// SIMATIC STEP 7 (V5.x) project BIW01_2012
// CPU: CPU 416-2 DP
// station: Hardware
// station: PLC1
// station: P_ADR_BUS
// program: GCPRO_Import
// program: Current400
// program: tmpGP-BIB
// program: tmpMH-BIB
// program: Current
// program: S7-Programm
// program: Baustein Kopie
// program: AG_Abzug
// program: temp
// program: temp2

SYMBOL_TABLE
"SYS_CBitDB"	DB 2	DB 2	// SYS: Changebit interface
"SYS_DirectCtrlDB"	DB 3	DB 3	// GCS7: PC direct control interface default DB
"SYS_HornDB"	DB 4	DB 4	// GCS7: Data Horn Modul
"SYS_LOG_Queue"	DB 5	DB 5	// PC Interface to log
"GCS7_GrCtrlDBTmp"	DB 6	FB 9	// Class date of FB9
"GCS7_RS485CtrlDB"	DB 7	FB 7	// GCS7: Communication controller opto22
"GCS7_ScaleControlDB"	DB 8	DB 8	// GCS7: Scale control buffer
"GCS7_GrCtrlDB"	DB 9	DB 9	// GCS7: Group control buffer
"SYS_DirectCtrlLCDB"	DB 10	DB 10	// GCS7: PC Direct Control Interface Remote Parameter
"TEST_IOSimuliInput"	DB 16	DB 16	// TEST: Only for serial (MPI) simulation
"TEST_IOSimuliOutput"	DB 17	DB 17	// TEST: Only for serial (MPI) simulation
"KebaHT4Data"	DB 20	FB 80	// Data KebaHT4Data
"SYS_PCCDirectCtrlDB"	DB 40	DB 40	// SYS: PC direct control interface PIC / WinCos /MELE
"SYS_PC1DirectCtrlDB"	DB 41	DB 41	// SYS: PC direct control interface pcc 1 (WinCC)
"SYS_PC2DirectCtrlDB"	DB 42	DB 42	// SYS: PC direct control interface pcc 2 (WinCC)
"SYS_PC3DirectCtrlDB"	DB 43	DB 43	// SYS: PC direct control interface pcc 1 (WinCC)
"SYS_PC4DirectCtrlDB"	DB 44	DB 44	// SYS: PC direct control interface pcc 4 (WinCC)
"SYS_PC5DirectCtrlDB"	DB 45	DB 45	// SYS: PC direct control interface pcc 5 (WinCC)
"SYS_PC6DirectCtrlDB"	DB 46	DB 46	// SYS: PC direct control interface pcc 6 (WinCC)
"SYS_PC7DirectCtrlDB"	DB 47	DB 47	// SYS: PC direct control interface pcc 7 (WinCC)
"SYS_ObjViewDirectCtrlDB"	DB 48	DB 48	// SYS: PC direct control interface for ObjView
"SYS_IHTestDirectCtrlDB"	DB 49	DB 49	// SYS: PC direct control interface for inhouse test
"PLC_SystemDB"	DB 50	DB 50	// PLC: System informations
"PLC_DPInfo"	DB 51	DB 51	// Summary Slave errors
"SSA_SYS_ASI_Info"	DB 52	DB 52	// Summary Slave errors
"PC_StorageDB"	DB 53	DB 53	// PC: Storage with free assignment
"ASW_TimerSettings"	DB 56	DB 56	// ASW: Timer settings
"ASW_Counter"	DB 57	DB 57	// ASW: Counter presettings
"SYS_PC1CBitDB"	DB 61	UDT 10020	// SYS: Changebit interface pcc 1 | PIC.LCT | MELE
"SYS_PC2CBitDB"	DB 62	UDT 10020	// SYS: Changebit interface pcc 2 | PIC.LMX
"SYS_PC3CBitDB"	DB 63	UDT 10020	// SYS: Changebit interface pcc 3
"SYS_PC4CBitDB"	DB 64	UDT 10020	// SYS: Changebit interface pcc 4
"GCS7_EREDB"	DB 71	FB 71	// GCS7: ERE
"SYS_DPInfoM1"	DB 75	FB 76	// SYS: PROFIBUS-DP diagnostic master 1
"SYS_DPInfoM2"	DB 76	FB 76	// SYS: PROFIBUS-DP diagnostic master 2
"SYS_DPInfoM3"	DB 77	FB 76	// SYS: PROFIBUS-DP diagnostic master 3
"SYS_DPInfoM4"	DB 78	FB 76	// SYS: PROFIBUS-DP diagnostic master 4
"PLC_BinListDB"	DB 79	FB 79	// Central bin list DB
"ASW_GraphicData"	DB 80	DB 80	// Win CC animation: Ways, function key, plant parameter
"ASW_PlantParData"	DB 81	DB 81	// Plant parameters and data time
"PCC_Data4"	DB 84	DB 84	// WinCC/PIC
"PCC_Data5"	DB 85	DB 85	// WinCC/PIC
"PCC_Data6"	DB 86	DB 86	// WinCC/PIC
"PCC_Data7"	DB 87	DB 87	// WinCC/PIC
"PCC_Data8"	DB 88	DB 88	// WinCC/PIC
"PCC_Data9"	DB 89	DB 89	// WinCC/PIC
"PCC_YieldScaleDB"	DB 90	DB 90	// PCC: Databuffer for PCC yield calculation
"COM_RS485Loop1DB"	DB 91	FB 7	// COM: RS485 loop1 scales and MYEB
"COM_RS485Loop2DB"	DB 92	FB 7	// COM: RS485 loop2 roolers
"COM_RS485Loop3DB"	DB 93	FB 7	// COM: RS485 loop3
"COM_RS485Loop4DB"	DB 94	FB 7	// COM: RS485 loop4
"SYS_SimpleDPInfo4DB"	DB 98	DB 98	// Data DP Diagnose
"SYS_StartWarningDB"	DB 100	FB 100	// SYS:  Startwarning modul
"ASW_DFCATargData"	DB 480	DB 480	// ASW_DFCATargData
"PLC1Snd"	DB 1711	DB 1711	// COM: Send data to PLC 1
"PLC2Snd"	DB 1712	DB 1712	// COM: Send data to PLC 2
"PLC3Snd"	DB 1713	DB 1713	// COM: Send data to PLC 3
"PLC4Snd"	DB 1714	DB 1714	// COM: Send data to PLC 4
"PLC5Snd"	DB 1715	DB 1715	// COM: Send data to PLC 5
"PLC6Snd"	DB 1716	DB 1716	// COM: Send data to PLC 6
"PLC7Snd"	DB 1717	DB 1717	// COM: Send data to PLC 7
"PLC8Snd"	DB 1718	DB 1718	// COM: Send data to PLC 8
"PLC9Snd"	DB 1719	DB 1719	// COM: Send data to PLC 9
"PLC1Rcv"	DB 1721	DB 1721	// COM: Receive data from PLC 1
"PLC2Rcv"	DB 1722	DB 1722	// COM: Receive data from PLC 2
"PLC3Rcv"	DB 1723	DB 1723	// COM: Receive data from PLC 3
"PLC4Rcv"	DB 1724	DB 1724	// COM: Receive data from PLC 4
"PLC5Rcv"	DB 1725	DB 1725	// COM: Receive data from PLC 5
"PLC6Rcv"	DB 1726	DB 1726	// COM: Receive data from PLC 6
"PLC7Rcv"	DB 1727	DB 1727	// COM: Receive data from PLC 7
"PLC8Rcv"	DB 1728	DB 1728	// COM: Receive data from PLC 8
"PLC9Rcv"	DB 1729	DB 1729	// COM: Receive data from PLC 9
"PLC10Snd"	DB 1730	DB 1730	// COM: Send data to PLC 10
"PLC11Snd"	DB 1731	DB 1731	// COM: Send data to PLC 11
"PLC12Snd"	DB 1732	DB 1732	// COM: Send data to PLC 12
"PLC13Snd"	DB 1733	DB 1733	// COM: Send data to PLC 13
"PLC14Snd"	DB 1734	DB 1734	// COM: Send data to PLC 14
"PLC15Snd"	DB 1735	DB 1735	// COM: Send data to PLC 15
"PLC16Snd"	DB 1736	DB 1736	// COM: Send data to PLC 16
"PLC10Rcv"	DB 1740	DB 1740	// COM: Receive data from PLC 10
"PLC11Rcv"	DB 1741	DB 1741	// COM: Receive data from PLC 11
"PLC12Rcv"	DB 1742	DB 1742	// COM: Receive data from PLC 12
"PLC13Rcv"	DB 1743	DB 1743	// COM: Receive data from PLC 13
"PLC14Rcv"	DB 1744	DB 1744	// COM: Receive data from PLC 14
"PLC15Rcv"	DB 1745	DB 1745	// COM: Receive data from PLC 15
"PLC16Rcv"	DB 1746	DB 1746	// COM: Receive data from PLC 16
"ComPLC1Snd"	DB 1761	FB 1701	// COM: Send buffer PLC 1
"ComPLC2Snd"	DB 1762	FB 1701	// COM: Send buffer PLC 2
"ComPLC3Snd"	DB 1763	FB 1701	// COM: Send buffer PLC 3
"ComPLC4Snd"	DB 1764	FB 1701	// COM: Send buffer PLC 4
"ComPLC5Snd"	DB 1765	FB 1701	// COM: Send buffer PLC 5
"ComPLC6Snd"	DB 1766	FB 1701	// COM: Send buffer PLC 6
"ComPLC7Snd"	DB 1767	FB 1701	// COM: Send buffer PLC 7
"ComPLC8Snd"	DB 1768	FB 1701	// COM: Send buffer PLC 8
"ComPLC9Snd"	DB 1769	FB 1701	// COM: Send buffer PLC 9
"ComPLC1Rcv"	DB 1771	FB 1702	// COM: Receive buffer PLC 1
"ComPLC2Rcv"	DB 1772	FB 1702	// COM: Receive buffer PLC 2
"ComPLC3Rcv"	DB 1773	FB 1702	// COM: Receive buffer PLC 3
"ComPLC4Rcv"	DB 1774	FB 1702	// COM: Receive buffer PLC 4
"ComPLC5Rcv"	DB 1775	FB 1702	// COM: Receive buffer PLC 5
"ComPLC6Rcv"	DB 1776	FB 1702	// COM: Receive buffer PLC 6
"ComPLC7Rcv"	DB 1777	FB 1702	// COM: Receive buffer PLC 7
"ComPLC8Rcv"	DB 1778	FB 1702	// COM: Receive buffer PLC 8
"ComPLC9Rcv"	DB 1779	FB 1702	// COM: Receive buffer PLC 9
"ComPLC10Snd"	DB 1780	FB 1701	// COM: Send buffer PLC 10
"ComPLC11Snd"	DB 1781	FB 1701	// COM: Send buffer PLC 11
"ComPLC12Snd"	DB 1782	FB 1701	// COM: Send buffer PLC 12
"ComPLC13Snd"	DB 1783	FB 1701	// COM: Send buffer PLC 13
"ComPLC14Snd"	DB 1784	FB 1701	// COM: Send buffer PLC 14
"ComPLC15Snd"	DB 1785	FB 1701	// COM: Send buffer PLC 15
"ComPLC16Snd"	DB 1786	FB 1701	// COM: Send buffer PLC 16
"ComPLC10Rcv"	DB 1790	FB 1702	// COM: Receive buffer PLC 7
"ComPLC11Rcv"	DB 1791	FB 1702	// COM: Receive buffer PLC 1
"ComPLC12Rcv"	DB 1792	FB 1702	// COM: Receive buffer PLC 2
"ComPLC13Rcv"	DB 1793	FB 1702	// COM: Receive buffer PLC 3
"ComPLC14Rcv"	DB 1794	FB 1702	// COM: Receive buffer PLC 4
"ComPLC15Rcv"	DB 1795	FB 1702	// COM: Receive buffer PLC 5
"ComPLC16Rcv"	DB 1796	FB 1702	// COM: Receive buffer PLC 6
"SSA_VIS_Filter"	DB 2010	DB 2010	// Filter DB to convert Status for Viscontrol
"SIEMENS_READ"	FB 3	FB 3	// SIEMENS: FMS.read services with SIMATIC NET CPs
"SIEMENS_WRITE"	FB 6	FB 6	// SIEMENS: FMS.write services with SIMATIC NET CPs
"GCS7_RS485Ctrl"	FB 7	FB 7	// GCS7: Communication controller opto22
"GCS7_GrpCtrlMain"	FB 9	FB 9	// GCS7: Group control main program
"GCS7_GrpCtrlSub"	FB 10	FB 10	// GCS7: Group control subroutines
"GCS7_E_DigOutput"	FB 11	FB 11	// GCS7: Element digital output
"GCS7_E_Motor"	FB 12	FB 12	// GCS7: Element motor
"GCS7_E_ValveControl"	FB 13	FB 13	// GCS7: Element valve control
"GCS7_E_DigInput"	FB 14	FB 14	// GCS7: Element digital input continuous
"GCS7_E_PressureRange"	FB 16	FB 16	// GCS7: Element pressure range
"GCS7_E_AnalogOutput"	FB 17	FB 17	// GCS7: Element analog output
"GCS7_E_ATV"	FB 18	FB 18	// Element Control FU Altivar with Profibus
"GCS7_E_AnalogInput"	FB 19	FB 19	// GCS7: Element analog input
"GCS7_E_ValveControl4Pos"	FB 20	FB 20	// GCS7: Element valve control with 4 positions
"GCS7_E_DMDS"	FB 21	FB 21	// GCS7: Element DMDS
"GCS7_E_MZMN"	FB 22	FB 22	// GCS7: Element MZMN micro dosing
"GCS7_E_MYEB"	FB 23	FB 23	// GCS7: Element MYEB moisture control unit
"GCS7_E_MOZE"	FB 24	FB 24	// GCS7: Element MOZE water doser
"GCS7_E_MessageCtrl"	FB 25	FB 25	// GCS7: Element Control Message
"GCS7_E_DFCO"	FB 26	FB 26
"GCS7_E_MEAF_Bag"	FB 27	FB 27	// GCS7: Element Control MEAF-Bag with DP or OPTO22
"GCS7_E_FBAL"	FB 28	FB 28	// GCS7: Element Control Message
"GCS7_E_Sampler"	FB 29	FB 29	// GCS7: Element sampler MZER
"GCS7_E_Maintanance1"	FB 30	FB 30	// GCS7: Element Control Message
"GCS7_E_Maintanance2"	FB 31	FB 31	// GCS7: Element Control Message
"GCS7_E_MZAF"	FB 32	FB 32	// GCS7: Element MZAF flowbalancer
"GCS7_E_MYAH"	FB 33	FB 33	// GCS7: Element MYAH Yield PC
"GCS7_E_MYFC_MOZF"	FB 34	FB 34	// GCS7: Element MYFC/MOZF
"GCS7_E_MDDx"	FB 35	FB 35	// GCS7 Element MDDx Opto22 Communication
"GCS7_E_MYRA_MDEx"	FB 36	FB 36	// GCS7: Element MYRA/MDEF
"GCS7_E_MDDx_DP"	FB 37	FB 37	// SSW: Element MDDR/T Profibus Communication
"GCS7_E_DEVC"	FB 38	FB 38	// GCS7: Element MEAF Dev Control
"GCS7_E_MYFA_MOZD"	FB 39	FB 39	// GCS7: Element MYFA/MOZD automatic dampener
"GCS7_E_Scale"	FB 40	FB 40	// GCS7: Element scale control MWEE, MWEG,
"GCS7_M_MYFA"	FB 41	FB 41	// GCS7: Machine MYFA
"GCS7_E_BSPB"	FB 42	FB 42	// Vertikalschleifer
"GCS7_E_DCOS"	FB 43	FB 43	// GCS7: Element Control Dosing Control System
"GCS7_M_Scourer"	FB 44	FB 44	// GCS7: Machine scourer MHXF
"GCS7_M_Roll4Stand"	FB 45	FB 45	// GCS7: Machine 4 roll stand
"GCS7_M_Roll8Stand"	FB 46	FB 46	// GCS7: Machine 8 roll stand
"GCS7_M_PelletCooler"	FB 47	FB 47	// GCS7: Machine pellet cooler
"GCS7_M_Motors3W2HL"	FB 48	FB 48	// GCS7: Machine 3 Motors and 2 high levels
"GCS7_M_MDDX"	FB 49	FB 49	// GCS7: Machine Newtronic Roll Stand
"GCS7_M_Motor6Mon"	FB 50	FB 50	// GCS7: Machine motor with 6 monitoring elements
"GCS7_M_Motor2Mon"	FB 51	FB 51	// GCS7: Machine motor with 2 monitoring elements
"GCS7_M_MotorBypass"	FB 52	FB 52	// GCS7: Machine motor with bypass
"GCS7_M_Hopper"	FB 53	FB 53	// GCS7: Machine hopper
"GCS7_M_Mixer"	FB 54	FB 54	// GCS7: Machine mixer
"GCS7_M_DFZK"	FB 55	FB 55	// GCS7 Machine DFZK Vertical Rotor Mill
"GCS7_M_Discharger"	FB 56	FB 56	// GCS7: Machine discharger A
"GCS7_E_MTRI"	FB 57	FB 57	// GCS7: Element MTRI Remote Control
"GCS7_M_BCFA"	FB 58	FB 58	// GCS7: Machine Flaker Control System
"GCS7_M_DischargerMZAx"	FB 59	FB 59	// GCS7: Machine discharger with MZAF
"GCS7_M_Aspiration"	FB 60	FB 60	// GCS7: Machine aspiration
"GCS7_M_DPScaleMWBL_MWBS"	FB 61	FB 61	// GCS7: Machine MWBL/MWBS (Profibus+ Opto22)
"GCS7_M_DriveCurrent"	FB 62	FB 62	// GCS7: Machine DriveCurrent
"GCS7_M_DFCA"	FB 63	FB 63	// GCS7: Machine DFCA
"GCS7_M_MYFB"	FB 64	FB 64	// GCS7: Machine MYFB automatic dampener
"GCS7_M_PulsePhaseConv"	FB 65	FB 65	// GCS7: Machine pulse phase conveying system
"GCS7_M_Flift1Airlock"	FB 66	FB 66	// GCS7: Machine fluidlift with 1 airlock
"GCS7_M_Flift2Airlock"	FB 67	FB 67	// GCS7: Machine fluidlift with 2 airlocks
"GCS7_M_PressureVessel"	FB 68	FB 68	// GCS7 Machine Pressure Vessel Conveying
"GCS7_M_RotaryDis"	FB 69	FB 69	// GCS7: Machine rotary distributer
"GCS7_AddWayPattern"	FB 70	FB 70	// GCS7: Old and new waypattern are active
"GCS7_E_MaintananceCnt"	FB 71	FB 71	// GCS7: Maintanance Counter
"GCS7_E_DFCA_Com"	FB 73	FB 73	// GCS7: Communication DFCA pellet press
"GCS7_E_DFCA_Log"	FB 74	FB 74	// GCS7: Log when modify a parameter
"SYS_DP-Diagnosis"	FB 76	FB 76	// SIEMENS_DP-Diagnosis
"GCS7_ULQueue"	FB 77	FB 77
"GCS7_Bin"	FB 78	FB 78	// Functionality of a bin
"PLC_BinList"	FB 79	FB 79	// Central bin list
"KebaHT4"	FB 80	FB 80	// MAINTENANCE MOTOR CONTROL "HT4"
"GCS7_M_RGRP"	FB 81	FB 81	// GCS7: Machine RGRP
"GCS7_M_FluidlifVessel"	FB 82	FB 82	// GCS7 Machine Fluidlift with Pressure Vessel
"GCS7_E_Level"	FB 84	FB 84	// Level: Subtype of FB14
"GCS7_LiftingDevice"	FB 85	FB 85	// de: Hubzug
"GCS7_TractionDrive"	FB 86	FB 86	// Traction drive  de: Fahrantrieb
"GCS7_M_Roll8Stand_DP"	FB 87	FB 87	// SS: Machine 4/8 roll stand wit profibus
"GCS7_Ma_DischagerFlat"	FB 88	FB 88	// Machine Flat-bottom discharger
"STD_LineSecStdSub2"	FB 90	FB 90	// STD: Line and section control standard subroutines
"SYS_DPMultiDPInfo"	FB 98	FB 98	// SimpleMultiDPInfo
"SYS_DPDiagnostic"	FB 99	FB 99	// SYS: DP diagnostic and monitoring
"GCS7_StartWarning"	FB 100	FB 100	// GCS7 Start Warning Modul
"Gr050_Code"	FB 150	FB 150	// Group-FB  Machine FB44, FB47, FB50, FB51, FB52, FB56
"STD_StartupBinTime"	FB 801	FB 801	// STD: Startup bin filling procedure
"SSA_PneumaticControl_Fct"	FB 841	FB 841	// SSA: Pneumatic controller
"SSW_EL_ASI_Fct"	FB 899	FB 899	// Element Control ASI Master Wago/Profibus
"COM_PLCSend"	FB 1701	FB 1701	// COM: Send data to an other PLC
"COM_PLCReceive"	FB 1702	FB 1702	// COM: Receive data from an other PLC
"STD_PLCWatchdog"	FB 1703	FB 1703	// STD: PLC to PLC communication watchdog
"COM_Modbus_CMV96"	FB 1709	FB 1709	// Modbus interface to CMV96
"SSA_EL_Sampler_RFID"	FB 1714	FB 1714	// Baumer RFID
"SYS_CBitCtrl"	FC 2	FC 2	// SYS: Call change bit controller
"SYS_DirectCtrl"	FC 3	FC 3	// GCS7: PC direct control subroutines
"SYS_Horn_Code"	FC 4	FC 4	// GCS7: Code Horn Modul
"AG_SEND"	FC 5	FC 5	// Send Function for SEND-/RECEIVE-Services to SIMATIC NET CPs
"AG_RECEIVE"	FC 6	FC 6	// Receive Function for SEND-/RECEIVE-Services to SIMATIC NET CPs
"SYS_CallGroup"	FC 9	FC 9	// SYS: Call group functions blocks
"ASW_SimulElements"	FC 10	FC 10	// USW: Element simulation
"SYS_CallLineSection"	FC 11	FC 11	// SYS: Call line and section controller
"SYS_RW_IO"	FC 12	FC 12	// SYS: Read/Write IO of elements
"TEST_IOSIMULI_Copy"	FC 16	FC 16	// TEST: Functions for serial IO-Manager
"GCS7_TON_LONG"	FC 17	FC 17	// Timer TON long time values
"GCS7_TON"	FC 18	FC 18	// Timer TON
"SYS_Analog_S5_to_S7"	FC 19	FC 19	// Convert analog value S5 format to S7 for
"CWA_ScaleSimul"	FC 39	FC 39	// CWA: Scale simulation
"CWA_ScaleCtrlSub"	FC 40	FC 40	// CWA: Scale control subroutines
"CWA_ScaleCtrlMain"	FC 41	FC 41	// CWA: Scale control main program
"CWA_ScaleRead"	FC 42	FC 42	// CWA: Scale read
"GCS7_LogConvert"	FC 45	FC 45	// LOG: GCS7 message convert
"SYS_LOG_EntryQueue"	FC 46	FC 46	// LOG: Message entry in queue
"SYS_LOG_CtrlQueue"	FC 47	FC 47	// LOG: Call queue controller
"SYS_Copy_DBtoDB"	FC 49	FC 49	// SYS: Block transfer DB to DB
"SYS_Copy_Array_Element"	FC 50	FC 50
"SYS_DeleteDB"	FC 51	FC 51	// BASIS: Delete data block
"SYS_InitFlagTimer"	FC 52	FC 52	// SYS: Init flags and timers
"SYS_BitAddress"	FC 53	FC 53	// Get Bit Adress of any Symbol
"GCS7_LineCtrlMain"	FC 58	FC 58	// GCS7: Line control main program
"GCS7_LineCtrlSub"	FC 59	FC 59	// GCS7: Line control subroutines
"GCS7_SecCtrlMain"	FC 60	FC 60	// GCS7: Section control main program
"GCS7_SecCtrlSub"	FC 61	FC 61	// GCS7: Section control subroutines
"GCS7_SecCtrlASW"	FC 63	FC 63	// GCS7: Section control ASW subroutines
"GCS7_BinCtrlMain"	FC 66	FC 66	// GCS7: Bin control main program
"GCS7_BinCtrlSub"	FC 67	FC 67	// GCS7: Scale control subroutines
"GCS7_ScaleCtrlMain"	FC 68	FC 68	// GCS7: Scale control main program
"GCS7_ScaleCtrlSub"	FC 69	FC 69	// GCS7: Scale control subroutines
"GCS7_LogConvert_10"	FC 73	FC 73	// LOG: GCS7 message convert Format 10
"SYS_DPDiagMain"	FC 75	FC 75	// DPDiagnose Main program
"SYS_DPDiag1"	FC 76	FC 76	// DPDiagnose => not Siemens Slave
"GCS7BinCtrlUpdataLevel"	FC 78	FC 78	// GCS7: Bin Control Update Bin Level
"ASW_GraphicFunction"	FC 80	FC 80	// ASW: Preparation of fast values for visualisation
"ASW_PlantParFunction"	FC 81	FC 81	// ASW: Preparation of fast values for visualisation
"SIEMENS_IECFC6_DT_DATE"	FC 90	FC 90	// SIEMENS: Date from DATE_AND_TIME
"SIEMENS_IECFC8_DT_TOD"	FC 91	FC 91	// SIEMENS: Time from DATE_AND_TIME
"SIEMENS_IECFC3_D_TOD_DT"	FC 92	FC 92	// SIEMENS: DATE+TIME_OF_DAY --> DATE_AND_TIME
"SIEMENS_IECFC10_EQ_STR"	FC 93	FC 93	// SIEMENS: String Compare
"SYS_SimpleDPInfo"	FC 98	FC 98	// SYS: PROFIBUS-DP diagnostic
"SIEMENS_GlobalDPInfo"	FC 99	FC 99	// SIEMENS: PROFIBUS-DP monitoring
"SYS_GeneralPLCStartup"	FC 100	FC 100	// SYS: General plc startup functions
"SYS_GeneralFunctions"	FC 105	FC 105	// SYS: General plant signals
"HW_PanelLamps"	FC 106	FC 106	// HW: Lamps on control panel
"ConvertGrayCode"	FC 108	FC 108	// Convert Gray Code
"SSA_Analog_S5_to_S7"	FC 109	FC 109	// Convert analog value S5 format to S7 for
"TEST_Functions"	FC 111	FC 111	// TEST: Testfunctions
"STD_LineSecStdSub"	FC 120	FC 120	// STD: Line and section control standard subroutines
"STD_OnOffSignals"	FC 121	FC 121	// STD: ON / OFF Signal handling
"STD_OnOffSignals32"	FC 122	FC 122	// STD: ON / OFF Signal handling with 32-Bit
"COM_PLCtoPLC"	FC 141	FC 141	// COM: PLC to PLC communication
"VDU_MsgQueueEntry"	FC 145	FC 145	// VDU: Message entry into queue
"USW_CWAFastOperations"	FC 151	FC 151	// USW: Fast CWA operation, called by interrupt ob
"STD_SearchChangeBit"	FC 241	FC 241	// STD: Search object change bits
"STD_PLCLiveValue"	FC 242	FC 242	// STD: Live value handling for PCC
"STD_MinMaxSearch"	FC 243	FC 243	// STD: Search for min/max values
"STD_AuxiliaryFunctions"	FC 247	FC 247	// STD: Auxiliary functions
"STD_QueueManager"	FC 251	FC 251	// STD: Queue manager main program
"STD_QueueSub"	FC 252	FC 252	// STD: Queue manager sub program copy/search
"STD_QueueIdx"	FC 253	FC 253	// STD: Queue manager sub program index
"STD_QueueFilter"	FC 254	FC 254	// STD: Queue manager sub program compare
"STD_QueueModEntry"	FC 256	FC 256	// STD: Queue manager log queue entry
"ASW_StageCtrl_Fct"	FC 1800	FC 1800
"SSA_Vis_Update"	FC 2042	FC 2042	// Update Handshake for Graphik Update
"SSA_VIS_Status"	FC 2043	FC 2043	// Convert Status for Viscontrol
"SSA_VIS_Log_Msg"	FC 2055	FC 2055	// Enter Viscontrol Log Message
"CPU_CopyPulse100ms"	M 1.0	BOOL	// CPU: System timing
"CPU_CopyPulse200ms"	M 1.1	BOOL	// CPU: System timing
"CPU_CopyPulse400ms"	M 1.2	BOOL	// CPU: System timing
"CPU_CopyPulse500ms"	M 1.3	BOOL	// CPU: System timing
"CPU_CopyPulse800ms"	M 1.4	BOOL	// CPU: System timing
"CPU_CopyPulse1000ms"	M 1.5	BOOL	// CPU: System timing
"CPU_CopyPulse1600ms"	M 1.6	BOOL	// CPU: System timing
"CPU_CopyPulse1800ms"	M 1.7	BOOL	// CPU: System timing
"CPU_Pulse100ms"	M 2.0	BOOL	// CPU: System timing
"CPU_Pulse200ms"	M 2.1	BOOL	// CPU: System timing
"CPU_Pulse400ms"	M 2.2	BOOL	// CPU: System timing
"CPU_Pulse500ms"	M 2.3	BOOL	// CPU: System timing
"CPU_Pulse800ms"	M 2.4	BOOL	// CPU: System timing
"CPU_Pulse1000ms"	M 2.5	BOOL	// CPU: System timing
"CPU_Pulse1600ms"	M 2.6	BOOL	// CPU: System timing
"CPU_Pulse2000ms"	M 2.7	BOOL	// CPU: System timing
"SYS_ScanA_IsOn"	M 3.1	BOOL	// SYS: Scan A is active
"SYS_ScanB_IsOn"	M 3.2	BOOL	// SYS: Scan B is active
"SYS_ScanC_IsOn"	M 3.3	BOOL	// SYS: Scan C is active
"Sys_Tick100msFromFastOB"	M 3.6	BOOL
"Sys_Tick200msFromFastOB"	M 3.7	BOOL
"SYS_Scan0_Tick100ms"	M 4.2	BOOL	// SYS_Scan0: Is every 100ms for one scan high
"SYS_Scan0_Tick200ms"	M 4.3	BOOL	// SYS_Scan0: Is every 200ms for one scan high
"SYS_Scan0_Tick500ms"	M 4.4	BOOL	// SYS_Scan0: Is every 500ms for one scan high
"SYS_Scan0_Tick1s"	M 4.5	BOOL	// SYS_Scan0: Is every 1s for one scan high
"SYS_Scan0_Tick1min"	M 4.6	BOOL	// SYS_Scan0: Is every min for one scan high
"SYS_ScanA_Tick200ms"	M 5.3	BOOL	// SYS_ScanA: Is every 200ms for one scan high
"SYS_ScanA_Tick500ms"	M 5.4	BOOL	// SYS_ScanA:  Is every 500ms for one scan high
"SYS_ScanA_Tick1s"	M 5.5	BOOL	// SYS_ScanA: Is every 1s for one scan high
"SYS_ScanA_Tick1min"	M 5.6	BOOL	// SYS_ScanA: Is every min for one scan high
"SYS_ScanB_Tick200ms"	M 6.3	BOOL	// SYS_ScanB: Is every 200ms for one scan high
"SYS_ScanB_Tick500ms"	M 6.4	BOOL	// SYS_ScanB: Is every 500ms for one scan high
"SYS_ScanB_Tick1s"	M 6.5	BOOL	// SYS_ScanB: Is every 1s for one scan high
"SYS_ScanB_Tick1min"	M 6.6	BOOL	// SYS_ScanB: Is every min for one scan high
"SYS_ScanC_Tick200ms"	M 7.3	BOOL	// SYS_ScanC: Is every 200ms for one scan high
"SYS_ScanC_Tick500ms"	M 7.4	BOOL	// SYS_ScanC: Is every 500ms for one scan high
"SYS_ScanC_Tick1s"	M 7.5	BOOL	// SYS_ScanC: Is every 1s for one scan high
"SYS_ScanC_Tick1min"	M 7.6	BOOL	// SYS_ScanC: Is every min for one scan high
"SYS_infLog0"	M 9.0	BOOL	// SYS: Logical false all the time
"SYS_infLog1"	M 9.1	BOOL	// SYS: Logical true all the time
"SYS_CycleFlasher"	M 9.2	BOOL	// SYS: Status changing every scan
"SYS_Pulse500ms"	M 9.3	BOOL	// SYS: Pulse 500 ms true, 500ms false
"SYS_Pulse1000ms"	M 9.4	BOOL	// SYS: Pulse 1000ms true, 1000ms false
"SYS_Tick1s"	M 9.5	BOOL	// SYS: Tick is every 1s for one scan high
"GCS7_Gr_OutTick100ms"	M 10.2	BOOL	// GCS7: Group control module
"GCS7_Gr_OutTick200ms"	M 10.3	BOOL	// GCS7: Group control module
"GCS7_Gr_OutTick500ms"	M 10.4	BOOL	// GCS7: Group control module
"GCS7_Gr_OutTick1s"	M 10.5	BOOL	// GCS7: Group control module
"GCS7_Gr_OutTick1min"	M 10.6	BOOL	// GCS7: Group control module
"GCS7_Gr_OutRestartPLC"	M 11.0	BOOL	// GCS7: Group control module
"GCS7_Gr_SimDPtoImage"	M 11.1	BOOL	// GCS7: 1=Simulator uses process image GCS7:  0=Simulator uses DB16/17
"GCS7_Gr_OutLogOff"	M 11.2	BOOL	// GCS7: Group control module
"GCS7_Gr_OutCallFast1"	M 11.4	BOOL	// GCS7: Group control module
"GCS7_Gr_OutCallFast2"	M 11.5	BOOL	// GCS7: Group control module
"GCS7_Gr_OutCallFast3"	M 11.6	BOOL	// GCS7: Group control module
"GCS7_Gr_InBrakeMill"	M 12.0	BOOL	// GCS7: Is set by DFCA, when any machine is stoppinf with brake
"GCS7_Gr_OutNext"	M 12.2	BOOL	// GCS7: Group control module
"GCS7_Gr_OutFaultReset"	M 12.3	BOOL	// GCS7: Group control module
"GCS7_Gr_OutManualOff"	M 12.4	BOOL	// GCS7: Group control module
"GCS7_Gr_OutManualOn"	M 12.5	BOOL	// GCS7: Group control module
"GCS7_Gr_OutReportAll"	M 12.6	BOOL	// GCS7: Group control module
"GCS7_Gr_InCBit1"	M 13.0	BOOL	// GCS7: Group control module
"GCS7_Gr_InCBit2"	M 13.1	BOOL	// GCS7: Group control module
"GCS7_Gr_InCBit3"	M 13.2	BOOL	// GCS7: Group control module
"GCS7_Gr_InCBit4"	M 13.3	BOOL	// GCS7: Group control module
"GCS7_Gr_InFault"	M 13.4	BOOL	// GCS7: Group control module
"GCS7_Gr_InManual"	M 13.5	BOOL	// GCS7: Group control module
"GCS7_Gr_InHeavyStartup"	M 13.6	BOOL	// GCS7: Group control module
"GCS7_Gr_InFaultFlag"	M 13.7	BOOL	// GCS7: Group control module
"GCS7_Gr_InHWStop"	M 15.0	BOOL	// GCS7: Group control module
"GCS7_Gr_InDPFault"	M 15.1	BOOL	// GCS7: Group control module
"GCS7_Gr_InForce"	M 15.3	BOOL	// GCS7: Group control module
"GCS7_Gr_InMaintWarning"	M 15.4	BOOL	// GCS7: Group control module - Any maintenance element has a warning
"GCS7_Gr_InMaintFault"	M 15.5	BOOL	// GCS7: Group control module - Any maintenance element has a fault
"ENG_RemarkFlag"	M 50.0	BOOL	// ENG: Remark to remove all that flags
"CPU_TimeFlagsCopy"	MB 1	BYTE	// CPU: System timing
"CPU_TimeFlags"	MB 2	BYTE	// CPU: System timing
"SYS_CyclePartioning"	MB 3	BYTE	// SYS: Cycle partitioning
"SYS_Scan0_Time"	MB 4	BYTE	// SYS_Scan0: Timer flag
"SYS_ScanA_Time"	MB 5	BYTE	// SYS_ScanA: Timer flag
"SYS_ScanB_Time"	MB 6	BYTE	// SYS_ScanB: Timer flag
"SYS_ScanC_Time"	MB 7	BYTE	// SYS_ScanC: Timer flag
"SYS_GeneralFlags"	MB 9	BYTE	// SYS: General flags
"GCS7_Gr_Tick"	MB 10	BYTE	// GCS7: Group control module
"GCS7_Gr_MainToElMa"	MB 11	BYTE	// GCS7: Information main prog. to element and machine
"GCS7_Gr_ElMaToGroup1"	MB 12	BYTE	// GCS7: Information Element and machine to group
"GCS7_Gr_ElMaToGroup2"	MB 13	BYTE	// GCS7: Information Element and machine to group
"GCS7_Gr_OutLine"	MB 14	BYTE	// GCS7: Group control module
"ENG_Settings"	MB 50	BYTE	// ENG: Engineering settings
"Gr_ParHornCode"	MW 16	WORD
"SYS_MainProgram"	OB 1	OB 1	// SYS: Main program
"SYS_TOD_INT1"	OB 10	OB 10	// SYS: Time of Day Interrupt 1
"SYS_TOD_INT2"	OB 11	OB 11	// SYS: Time of Day Interrupt 2
"SYS_DEL_INT1"	OB 20	OB 20	// SYS: Time Delay Interrupt 1
"SYS_DEL_INT2"	OB 21	OB 21	// SYS: Time Delay Interrupt 2
"SYS_CycInt5s"	OB 30	OB 30	// SYS: Cyclic interrupt 5 sec
"SYS_CycInt2s"	OB 31	OB 31	// SYS: Cyclic interrupt 2 sec
"SYS_CycInt500ms"	OB 33	OB 33	// SYS: Cyclic interrupt 500 ms
"SYS_CycInt200ms"	OB 34	OB 34	// SYS: Cyclic interrupt 200 ms
"SYS_CycInt20ms"	OB 35	OB 35	// SYS: Cyclic interrupt 20 ms
"SYS_CycInt50ms"	OB 36	OB 36	// SYS: Cyclic interrupt 50 ms
"SYS_CycInt100ms"	OB 37	OB 37	// SYS: Cyclic interrupt 100 ms
"SYS_CycInt10ms"	OB 38	OB 38	// SYS: Cyclic interrupt 10 ms
"SYS_HW_INT1"	OB 40	OB 40	// SYS: Hardware Interrupt 1
"SYS_HW_INT2"	OB 41	OB 41	// SYS: Hardware Interrupt 2
"SYS_CYCL_FLT"	OB 80	OB 80	// SYS: Cycle time fault
"SYS_PS_FLT"	OB 81	OB 81	// SYS: Power Supply Fault
"SYS_IO_FLT1"	OB 82	OB 82	// SYS: I/O Point Fault 1
"SYS_IO_FLT2"	OB 83	OB 83	// SYS: I/O Point Fault 2
"SYS_HW_CPUFault"	OB 84	OB 84	// HW: CPU hardware failure
"SYS_OBNL_FLT"	OB 85	OB 85	// SYS: OB Not Loaded Fault
"SYS_RACK_FLT"	OB 86	OB 86	// SYS: Loss of Rack Fault
"SYS_ComFailure"	OB 87	OB 87	// SYS: Communication Fault
"PLC_StUpNewstart"	OB 100	OB 100	// PLC: Startup program on newstart
"PLC_StUpRestart"	OB 101	OB 101	// PLC: Startup program on restart
"PLC_StUpColdstart"	OB 102	OB 102	// PLC: Startup program on coldstart
"SYS_PROG_ERR"	OB 121	OB 121	// SYS: Programming Error
"SYS_MOD_ERR"	OB 122	OB 122	// SYS: Module Access Error
"CTUD"	SFB 2	SFB 2	// Count Up / Down
"TON"	SFB 4	SFB 4	// Generate an On Delay
"SIEMENS_BSEND"	SFB 12	SFB 12	// SIEMENS: Block Oriented Send
"SIEMENS_BRCV"	SFB 13	SFB 13	// SIEMENS: Block Oriented Receive
"SIEMENS_HS_COUNT"	SFB 29	SFB 29	// SIEMENS: High-Speed Counter (CPU 312, Integrated Function)
"SIEMENS_FREQ_MES"	SFB 30	SFB 30	// SIEMENS: Frequency Meter (CPU 312, Integrated Function)
"SIEMENS_POSITION"	SFB 31	SFB 31	// SIEMENS: Open-Loop Positioning (CPU 312, Integrated Function)
"SIEMENS_SET_CLK"	SFC 0	SFC 0	// SIEMENS: Set System Clock
"SIEMENS_READ_CLK"	SFC 1	SFC 1	// SIEMENS: Read System Clock
"SIEMENS_SET_RTM"	SFC 2	SFC 2	// SIEMENS: Set Run-Time Meter
"SIEMENS_CTRL_RTM"	SFC 3	SFC 3	// SIEMENS: Start/Stop Run-Time Meter
"SIEMENS_READ_RTM"	SFC 4	SFC 4	// SIEMENS: Read Run-Time Meter
"GADR_LGC"	SFC 5	SFC 5	// Query Logical Address of a Channel
"RD_SINFO"	SFC 6	SFC 6	// Read OB Start Information
"DPNRM_DG"	SFC 13	SFC 13	// Read Diagnostic Data of a DP Slave
"SIEMENS_DPRD_DAT"	SFC 14	SFC 14	// SIEMENS: Read data for DP-Node
"SIEMENS_DPWR_DAT"	SFC 15	SFC 15	// SIEMENS: Write Data to DP-Node
"SIEMENS_BLKMOV"	SFC 20	SFC 20	// SIEMENS: Direct Word Move
"SIEMENS_FILL"	SFC 21	SFC 21	// SIEMENS: Initialize a memory area
"SIEMENS_CREAT_DB"	SFC 22	SFC 22	// SIEMENS: Create Data Block
"SIEMENS_TEST_DB"	SFC 24	SFC 24	// SIEMENS: Test DB
"SIEMENS_SET_TINT"	SFC 28	SFC 28	// SIEMENS: Set Time-of-Day Interrupt
"SIEMENS_CAN_TINT"	SFC 29	SFC 29	// SIEMENS: Cancel Time-of-Day Interrupt
"SIEMENS_ACT_TINT"	SFC 30	SFC 30	// SIEMENS: Activate Time-of-Day Interrupt
"SIEMENS_QRY_TINT"	SFC 31	SFC 31	// SIEMENS: Query Time-of-Day Interrupt
"SIEMENS_SRT_DINT"	SFC 32	SFC 32	// SIEMENS: Start Time-Delay Interrupt
"SIEMENS_CAN_DINT"	SFC 33	SFC 33	// SIEMENS: Cancel Time-Delay Interrupt
"SIEMENS_QRY_DINT"	SFC 34	SFC 34	// SIEMENS: Query Time-Delay Interrupt
"SIEMENS_MSK_FLT"	SFC 36	SFC 36	// SIEMENS: Mask synchronous faults
"SIEMENS_DMSK_FLT"	SFC 37	SFC 37	// SIEMENS: Unmask Synchronous Faults
"SIEMENS_READ_ERR"	SFC 38	SFC 38	// SIEMENS: Read Error Registers
"SIEMENS_DIS_IRT"	SFC 39	SFC 39	// SIEMENS: Disable Interrupt
"SIEMENS_EN_IRT"	SFC 40	SFC 40	// SIEMENS: Enable New Interrupts and Asynchronous Errors
"SIEMENS_DIS_AIRT"	SFC 41	SFC 41	// SIEMENS: Disable Alarm Interrupts
"SIEMENS_EN_AIRT"	SFC 42	SFC 42	// SIEMENS: Enable Alarm Interrupts
"SIEMENS_RE_TRIGR"	SFC 43	SFC 43	// SIEMENS: Retrigger Cycle Time Monitoring
"SIEMENS_REPL_VAL"	SFC 44	SFC 44	// SIEMENS: Replace Value
"SIEMENS_STP"	SFC 46	SFC 46	// SIEMENS: Change the CPU to STOP
"SIEMENS_WAIT"	SFC 47	SFC 47	// SIEMENS: Wait
"SIEMENS_LGC_GADR"	SFC 49	SFC 49	// SIEMENS:
"SIEMENS_RD_LGADR"	SFC 50	SFC 50	// SIEMENS:
"SIEMENS_RDSYSST"	SFC 51	SFC 51	// SIEMENS: Read System Status
"SIEMENS_WR_USMSG"	SFC 52	SFC 52	// SIEMENS: Write User Element in Diagnosis Buffer
"SIEMENS_WR_PARM"	SFC 55	SFC 55	// SIEMENS: Synchronous Write Parameter (MC7)
"SIEMENS_WR_DPARM"	SFC 56	SFC 56	// SIEMENS: Synchronous Write Parameter (SDB)
"SIEMENS_PARM_MOD"	SFC 57	SFC 57	// SIEMENS: Synchronous Write Static and Dynamic
"SIEMENS_WR_REC"	SFC 58	SFC 58	// SIEMENS: Write Data Record
"SIEMENS_RD_REC"	SFC 59	SFC 59	// SIEMENS: Read Data Record
"SIEMENS_AB_CALL"	SFC 63	SFC 63	// SIEMENS: Assembly Code Block (CPU 614)
"SIEMENS_TIME_TCK"	SFC 64	SFC 64	// SIEMENS: Time Tick
"SYS_PLCStartUpDelay"	T 10	TIMER	// SYS: Delay software enable after plc startup
"SYS_HWDelay"	T 11	TIMER	// SYS: Delay software enable after hardware stop
"SYS_T_LOGEntryDelay"	T 13	TIMER	// SYS: Delay log entrys after fuse tripped
"SYS_T_OfflineDelay"	T 14	TIMER	// SYS: Delay section staOffline
"SYS_T_NStartOfflineTime"	T 15	TIMER	// SYS: Offline time after a newstart
"SYS_DelayHeavyStartup"	T 16	TIMER	// SYS: Monitoring time to reset flag
"SYS_DelayBrakeMill"	T 17	TIMER	// SYS: Monitoring time to reset flag brake mill
"COM_T_PCCWatchdog"	T 20	TIMER	// COM: Communication monitoring to process control computer
"ASW_Flags_F0_F15"	UDT 1000	UDT 1000
"ASW_LineAnimation"	UDT 1001	UDT 1001
"ASW_UserSectionState"	UDT 1002	UDT 1002
"ASW_ProductInfo"	UDT 1003	UDT 1003
"SSA_HandAddInfo"	UDT 1004	UDT 1004
"ASW_DFCARecipe"	UDT 1005	UDT 1005
"UDTL01LineCmd"	UDT 3200	UDT 3200
"UDTL01SecData"	UDT 3202	UDT 3202
"UDTL01SecAc"	UDT 3203	UDT 3203
"UDTL01SecNom"	UDT 3204	UDT 3204
"ASW_CBitDeclaration"	UDT 10020	UDT 10020	// ASW: Declaration of change bit data blocks
"GCS7_UDT_Timer"	UDT 10180	UDT 10180	// Timer in DB
"CWA_UDT_Command"	UDT 10413	UDT 10413	// UDT Command  for CWA
"CWA_UDT_BinParaShort"	UDT 10418	UDT 10418	// UDT CWA bin parameter with minimum used parameter
"CWA_UDT_BinParaAll"	UDT 10419	UDT 10419	// UDT CWA bin parameter with all parameters
"GCS7_UDT_FunctionKey"	UDT 10601	UDT 10601	// GCS7: Upper Layer
"GCS7_UDT_FaultPattern"	UDT 10602	UDT 10602	// GCS7: Upper Layer
"GCS7_UDT_StatusPattern"	UDT 10603	UDT 10603	// Upper Layer
"GCS7_UDT_BINList1"	UDT 10660	UDT 10660	// GCS7: Binlist without WtActual and WtTarget
"GCS7_UDT_BINStatus"	UDT 10662	UDT 10662	// GCS7: Binstatus
"GCS7_UDT_BINList2"	UDT 10664	UDT 10664	// GCS7: Binlist with WtActual without WtTarget
"GCS7_UDT_BINList3"	UDT 10668	UDT 10668	// GCS7: Binlist with WtActual and WtTarget
"GCS7_UDT_ScaleControl"	UDT 10680	UDT 10680	// GCS7: Scale control
"ASW_StageCtrl"	UDT 18000	UDT 18000
"PCCYieldScale"	UDT 19000	UDT 19000	// USW: Struct for scales involved in yield calculation
"WinCoSYieldScale"	UDT 19001	UDT 19001	// USW: Struct for scales involved in yield calculation
"SamplerData"	UDT 19002	UDT 19002	// USW: Struct for sampler data
"BigBagData"	UDT 19003	UDT 19003	// Registration of big bag weight
"GCS7_FB9_Section"	UDT 20090	UDT 20090	// Group Control: Interface Section
"GCS7_GR_COM"	UDT 20097	UDT 20097	// GCS7 Data PLC Communication per group
"GCS90S7_FB9_Communicat"	UDT 20098	UDT 20098	// Communication PLC --PLC GCS7 to GCS90S7
"GCS7_FB9_Communication"	UDT 20099	UDT 20099	// Communication PLC --PLC
"GCS7_FB11_Communication"	UDT 20119	UDT 20119	// Communication PLC --PLC
"GCS7_FB12_Communication"	UDT 20129	UDT 20129	// Communication PLC --PLC
"GCS7_FB13_Communication"	UDT 20139	UDT 20139	// Communication PLC --PLC
"GCS7_FB14_Communication"	UDT 20149	UDT 20149	// Communication PLC --PLC
"GCS7_FB16_Communication"	UDT 20169	UDT 20169	// Communication PLC --PLC
"GCS7_FB37_DP_Alarm"	UDT 20373	UDT 20373	// SSW: Element MDDR/T Alarms
"GCS7_FB40_dynData"	UDT 20400	UDT 20400	// Lower Layer
"GCS7_M_FB41_Data"	UDT 20410	UDT 20410	// Lower Layer
"GCS7_M_FB44_Data"	UDT 20440	UDT 20440	// Lower Layer
"GCS7_M_FB45_Data"	UDT 20450	UDT 20450	// Lower Layer
"GCS7_M_FB46_Data"	UDT 20460	UDT 20460	// Lower Layer
"GCS7_M_FB47_Data"	UDT 20470	UDT 20470	// Lower Layer
"GCS7_M_FB48_Data"	UDT 20480	UDT 20480	// Lower Layer
"GCS7_M_FB49_Data"	UDT 20490	UDT 20490	// Lower Layer
"GCS7_M_FB50_Data"	UDT 20500	UDT 20500	// Lower Layer
"GCS7_M_FB51_Data"	UDT 20510	UDT 20510	// Lower Layer
"GCS7_M_FB52_Data"	UDT 20520	UDT 20520	// Lower Layer
"GCS7_M_FB53_Data"	UDT 20530	UDT 20530	// Lower Layer
"GCS7_M_FB54_Data"	UDT 20540	UDT 20540	// Lower Layer
"GCS7_M_FB55_Data"	UDT 20550	UDT 20550	// Lower Layer
"GCS7_M_FB56_Data"	UDT 20560	UDT 20560	// Lower Layer
"GCS7_M_FB58_Data"	UDT 20580	UDT 20580	// Lower Layer
"GCS7_M_FB59_Data"	UDT 20590	UDT 20590	// Lower Layer
"GCS7_M_FB60_Data"	UDT 20600	UDT 20600	// Lower Layer
"GCS7_M_FB61_Data"	UDT 20610	UDT 20610	// Lower Layer
"GCS7_M_FB62_Data"	UDT 20620	UDT 20620	// Lower Layer
"GCS7_M_FB63_Data"	UDT 20630	UDT 20630	// Lower Layer
"GCS7_M_FB64_Data"	UDT 20640	UDT 20640	// Lower Layer
"GCS7_M_FB65_Data"	UDT 20650	UDT 20650	// Lower Layer
"GCS7_M_FB66_Data"	UDT 20660	UDT 20660	// Lower Layer
"GCS7_M_FB67_Data"	UDT 20670	UDT 20670	// Lower Layer
"GCS7_M_FB68_Data"	UDT 20680	UDT 20680	// Lower Layer
"GCS7_M_FB69_Data"	UDT 20690	UDT 20690	// Lower Layer
"GCS7_E_FB73_A201"	UDT 20735	UDT 20735	// DFCA: Data Telegram A201:
"GCS7_M_FB81_Data"	UDT 20810	UDT 20810	// Lower Layer
"GCS7_M_FB82_Data"	UDT 20820	UDT 20820	// Lower Layer
"GCS7_FB84_Communication"	UDT 20849	UDT 20849	// Communication PLC --PLC
"GCS7_FB85_Data"	UDT 20850	UDT 20850	// Stroke Drive
"GCS7_FB85_Counter"	UDT 20851	UDT 20851	// Data of Increment counter
"GCS7_FB86_Data"	UDT 20860	UDT 20860
"GCS7_M_FB87_Data"	UDT 20870	UDT 20870	// Machine 4/8 roll stand with profibus
"GCS7_M_FB88_Data"	UDT 20880	UDT 20880	// Machin Flat-bottom discharger
"GR052_UDT"	UDT 21520	UDT 21520	// UDT way groupAspiration Flaps Bin 21 to 34 (Aspiration)
"SSW_EL_ASI_Slave"	UDT 28995	UDT 28995	// Element Control ASI Master Wago/Profibus Slave Data
"ASW_UDTOnOffCmd"	UDT 32700	UDT 32700
"ASW_UDTSecNom"	UDT 32701	UDT 32701	// Nominal value for section
"ASW_UDTSecAc"	UDT 32702	UDT 32702	// Actual values of section
"VAT99"	VAT 99	
END_SYMBOL_TABLE

TYPE "SSA_HandAddInfo"	// UDT 1004
VERSION : 0.1
  STRUCT
   HandAddNr : INT ;
   ProductIdent : STRING  [16 ] := 'ABCDEFGHIJKLMNOP';
   ProductName : STRING  [32 ] := 'ABCDEFGHIJKLMNOPQRSTUVWXYZ012345';
   Barcode : STRING  [32 ] := 'ABCDEFGHIJKLMNOPQRSTUVWXYZ012345';
   TargetWeight : DINT ;	//Target Weight [gr]
   Reserve : ARRAY  [92 .. 99 ] OF BYTE ;
  END_STRUCT ;	
END_TYPE

TYPE "UDTL01LineCmd"	// UDT 3200
VERSION : 0.1
  STRUCT
   Cmd08 : BOOL ;	//Not used
   Cmd09 : BOOL ;	//Not used
   Cmd10 : BOOL ;	//Not used
   Cmd11 : BOOL ;	//Not used
   Cmd12 : BOOL ;	//Not used
   Cmd13 : BOOL ;	//Not used
   Cmd14 : BOOL ;	//Not used
   Cmd15 : BOOL ;	//Not used
   CmdPulse00OverrideLL : BOOL ;	//Override sender low levels
   CmdPulse01 : BOOL ;	//Not used
   CmdPulse02 : BOOL ;	//Not used
   CmdPulse03 : BOOL ;	//Not used
   CmdPulse04 : BOOL ;	//Not used
   CmdPulse05 : BOOL ;	//Not used
   CmdPulse06 : BOOL ;	//Not used
   CmdPulse07 : BOOL ;	//Not used
  END_STRUCT ;	
END_TYPE

TYPE "UDTL01SecAc"	// UDT 3203
VERSION : 0.1
  STRUCT
   Par1On : STRUCT 	//Job parameter status
    StaOn08 : BOOL ;	//Not used
    StaOn09 : BOOL ;	//Not used
    StaOn10 : BOOL ;	//Not used
    StaOn11 : BOOL ;	//Not used
    StaOn12 : BOOL ;	//Not used
    StaOn13 : BOOL ;	//Not used
    StaOn14 : BOOL ;	//Not used
    StaOn15 : BOOL ;	//Not used
    StaOn00 : BOOL ;	//Not used
    StaOn01 : BOOL ;	//Not used
    StaOn02 : BOOL ;	//Not used
    StaOn03 : BOOL ;	//Not used
    StaOn04 : BOOL ;	//Not used
    StaOn05 : BOOL ;	//Not used
    StaOn06 : BOOL ;	//Not used
    StaOn07 : BOOL ;	//Not used
   END_STRUCT ;
   Par1Off : WORD ;	//not used
   Par2On : STRUCT 	//Job parameter status
    StaOn08 : BOOL ;	//Not used
    StaOn09 : BOOL ;	//Not used
    StaOn10 : BOOL ;	//Not used
    StaOn11 : BOOL ;	//Not used
    StaOn12 : BOOL ;	//Not used
    StaOn13 : BOOL ;	//Not used
    StaOn14 : BOOL ;	//Not used
    StaOn15 : BOOL ;	//Not used
    StaOn00 : BOOL ;	//Not used
    StaOn01 : BOOL ;	//Not used
    StaOn02 : BOOL ;	//Not used
    StaOn03 : BOOL ;	//Not used
    StaOn04 : BOOL ;	//Not used
    StaOn05 : BOOL ;	//Not used
    StaOn06 : BOOL ;	//Not used
    StaOn07 : BOOL ;	//Not used
   END_STRUCT ;
   Par2Off : WORD ;	//not used
   Par3On : STRUCT 	//Job parameter status
    StaOn08 : BOOL ;	//Not used
    StaOn09 : BOOL ;	//Not used
    StaOn10 : BOOL ;	//Not used
    StaOn11 : BOOL ;	//Not used
    StaOn12 : BOOL ;	//Not used
    StaOn13 : BOOL ;	//Not used
    StaOn14 : BOOL ;	//Not used
    StaOn15 : BOOL ;	//Not used
    StaOn00 : BOOL ;	//Not used
    StaOn01 : BOOL ;	//Not used
    StaOn02 : BOOL ;	//Not used
    StaOn03 : BOOL ;	//Not used
    StaOn04 : BOOL ;	//Not used
    StaOn05 : BOOL ;	//Not used
    StaOn06 : BOOL ;	//Not used
    StaOn07 : BOOL ;	//Not used
   END_STRUCT ;
   Par3Off : WORD ;	//not used
   Par4On : STRUCT 	//Job parameter status
    StaOn08 : BOOL ;	//Not used
    StaOn09 : BOOL ;	//Not used
    StaOn10 : BOOL ;	//Not used
    StaOn11 : BOOL ;	//Not used
    StaOn12 : BOOL ;	//Not used
    StaOn13 : BOOL ;	//Not used
    StaOn14 : BOOL ;	//Not used
    StaOn15 : BOOL ;	//Not used
    StaOn00 : BOOL ;	//Not used
    StaOn01 : BOOL ;	//Not used
    StaOn02 : BOOL ;	//Not used
    StaOn03 : BOOL ;	//Not used
    StaOn04 : BOOL ;	//Not used
    StaOn05 : BOOL ;	//Not used
    StaOn06 : BOOL ;	//Not used
    StaOn07 : BOOL ;	//Not used
   END_STRUCT ;
   Par4Off : WORD ;	//not used
   ValueNotUsed9 : INT ;	//Not used
   ValueNotUsed10 : INT ;	//Not used
  END_STRUCT ;	
END_TYPE

TYPE "UDTL01SecNom"	// UDT 3204
VERSION : 0.1
  STRUCT
   Par1On : STRUCT 	//Job parameters
    Cmd08 : BOOL ;	//Not used
    Cmd09 : BOOL ;	//Not used
    Cmd10 : BOOL ;	//Not used
    Cmd11 : BOOL ;	//Not used
    Cmd12 : BOOL ;	//Not used
    Cmd13 : BOOL ;	//Not used
    Cmd14 : BOOL ;	//Not used
    Cmd15 : BOOL ;	//Not used
    Cmd00 : BOOL ;	//Not used
    Cmd01 : BOOL ;	//Not used
    Cmd02 : BOOL ;	//Not used
    Cmd03 : BOOL ;	//Not used
    Cmd04 : BOOL ;	//Not used
    Cmd05 : BOOL ;	//Not used
    Cmd06 : BOOL ;	//Not used
    Cmd07 : BOOL ;	//Not used
   END_STRUCT ;
   Par1Off : STRUCT 	//Job parameters
    Cmd08 : BOOL ;	//Not used
    Cmd09 : BOOL ;	//Not used
    Cmd10 : BOOL ;	//Not used
    Cmd11 : BOOL ;	//Not used
    Cmd12 : BOOL ;	//Not used
    Cmd13 : BOOL ;	//Not used
    Cmd14 : BOOL ;	//Not used
    Cmd15 : BOOL ;	//Not used
    Cmd00 : BOOL ;	//Not used
    Cmd01 : BOOL ;	//Not used
    Cmd02 : BOOL ;	//Not used
    Cmd03 : BOOL ;	//Not used
    Cmd04 : BOOL ;	//Not used
    Cmd05 : BOOL ;	//Not used
    Cmd06 : BOOL ;	//Not used
    Cmd07 : BOOL ;	//Not used
   END_STRUCT ;
   Par2On : STRUCT 	//Job parameters
    Cmd08 : BOOL ;	//Not used
    Cmd09 : BOOL ;	//Not used
    Cmd10 : BOOL ;	//Not used
    Cmd11 : BOOL ;	//Not used
    Cmd12 : BOOL ;	//Not used
    Cmd13 : BOOL ;	//Not used
    Cmd14 : BOOL ;	//Not used
    Cmd15 : BOOL ;	//Not used
    Cmd00 : BOOL ;	//Not used
    Cmd01 : BOOL ;	//Not used
    Cmd02 : BOOL ;	//Not used
    Cmd03 : BOOL ;	//Not used
    Cmd04 : BOOL ;	//Not used
    Cmd05 : BOOL ;	//Not used
    Cmd06 : BOOL ;	//Not used
    Cmd07 : BOOL ;	//Not used
   END_STRUCT ;
   Par2Off : STRUCT 	//Job parameters
    Cmd08 : BOOL ;	//Not used
    Cmd09 : BOOL ;	//Not used
    Cmd10 : BOOL ;	//Not used
    Cmd11 : BOOL ;	//Not used
    Cmd12 : BOOL ;	//Not used
    Cmd13 : BOOL ;	//Not used
    Cmd14 : BOOL ;	//Not used
    Cmd15 : BOOL ;	//Not used
    Cmd00 : BOOL ;	//Not used
    Cmd01 : BOOL ;	//Not used
    Cmd02 : BOOL ;	//Not used
    Cmd03 : BOOL ;	//Not used
    Cmd04 : BOOL ;	//Not used
    Cmd05 : BOOL ;	//Not used
    Cmd06 : BOOL ;	//Not used
    Cmd07 : BOOL ;	//Not used
   END_STRUCT ;
   Par3On : STRUCT 	//Job parameters
    Cmd08 : BOOL ;	//Not used
    Cmd09 : BOOL ;	//Not used
    Cmd10 : BOOL ;	//Not used
    Cmd11 : BOOL ;	//Not used
    Cmd12 : BOOL ;	//Not used
    Cmd13 : BOOL ;	//Not used
    Cmd14 : BOOL ;	//Not used
    Cmd15 : BOOL ;	//Not used
    Cmd00 : BOOL ;	//Not used
    Cmd01 : BOOL ;	//Not used
    Cmd02 : BOOL ;	//Not used
    Cmd03 : BOOL ;	//Not used
    Cmd04 : BOOL ;	//Not used
    Cmd05 : BOOL ;	//Not used
    Cmd06 : BOOL ;	//Not used
    Cmd07 : BOOL ;	//Not used
   END_STRUCT ;
   Par3Off : STRUCT 	//Job parameters
    Cmd08 : BOOL ;	//Not used
    Cmd09 : BOOL ;	//Not used
    Cmd10 : BOOL ;	//Not used
    Cmd11 : BOOL ;	//Not used
    Cmd12 : BOOL ;	//Not used
    Cmd13 : BOOL ;	//Not used
    Cmd14 : BOOL ;	//Not used
    Cmd15 : BOOL ;	//Not used
    Cmd00 : BOOL ;	//Not used
    Cmd01 : BOOL ;	//Not used
    Cmd02 : BOOL ;	//Not used
    Cmd03 : BOOL ;	//Not used
    Cmd04 : BOOL ;	//Not used
    Cmd05 : BOOL ;	//Not used
    Cmd06 : BOOL ;	//Not used
    Cmd07 : BOOL ;	//Not used
   END_STRUCT ;
   Par4On : STRUCT 	//Job parameters
    Cmd08 : BOOL ;	//Not used
    Cmd09 : BOOL ;	//Not used
    Cmd10 : BOOL ;	//Not used
    Cmd11 : BOOL ;	//Not used
    Cmd12 : BOOL ;	//Not used
    Cmd13 : BOOL ;	//Not used
    Cmd14 : BOOL ;	//Not used
    Cmd15 : BOOL ;	//Not used
    Cmd00 : BOOL ;	//Not used
    Cmd01 : BOOL ;	//Not used
    Cmd02 : BOOL ;	//Not used
    Cmd03 : BOOL ;	//Not used
    Cmd04 : BOOL ;	//Not used
    Cmd05 : BOOL ;	//Not used
    Cmd06 : BOOL ;	//Not used
    Cmd07 : BOOL ;	//Not used
   END_STRUCT ;
   Par4Off : STRUCT 	//Job parameters
    Cmd08 : BOOL ;	//Not used
    Cmd09 : BOOL ;	//Not used
    Cmd10 : BOOL ;	//Not used
    Cmd11 : BOOL ;	//Not used
    Cmd12 : BOOL ;	//Not used
    Cmd13 : BOOL ;	//Not used
    Cmd14 : BOOL ;	//Not used
    Cmd15 : BOOL ;	//Not used
    Cmd00 : BOOL ;	//Not used
    Cmd01 : BOOL ;	//Not used
    Cmd02 : BOOL ;	//Not used
    Cmd03 : BOOL ;	//Not used
    Cmd04 : BOOL ;	//Not used
    Cmd05 : BOOL ;	//Not used
    Cmd06 : BOOL ;	//Not used
    Cmd07 : BOOL ;	//Not used
   END_STRUCT ;
   LineFlowrate : INT ;	//Line flowrate, for turnover only
   NotUsed1 : INT ;	//Not used
   NotUsed2 : WORD ;
   NotUsed3 : WORD ;
   NotUsed4 : WORD ;
   NotUsed5 : WORD ;
  END_STRUCT ;	
END_TYPE

TYPE "CWA_UDT_Command"	// UDT 10413
VERSION : 0.0
  STRUCT 	//Function key for CWA
   CmdAcceptWt : BOOL ;
   CmdAbortBatch : BOOL ;
   CmdAbortIngr : BOOL ;
   Cmd43 : BOOL ;
   Cmd44 : BOOL ;
   Cmd45 : BOOL ;
   Cmd46 : BOOL ;
   Cmd47 : BOOL ;
   CmdStartSingleIngr : BOOL ;
   CmdModifyBin : BOOL ;
   CmdFinalEmptying : BOOL ;
   CmdEmptyingInterm : BOOL ;
   CmdManualAddReady : BOOL ;
   CmdNextStep : BOOL ;
   CmdReset : BOOL ;
   CmdRetry : BOOL ;
   CmdRestDischargeOff : BOOL ;
   Cmd25 : BOOL ;
   Cmd26 : BOOL ;
   Cmd27 : BOOL ;
   Cmd28 : BOOL ;
   Cmd29 : BOOL ;
   Cmd30 : BOOL ;
   Cmd31 : BOOL ;
   CmdSingleIngrOff : BOOL ;
   CmdLogIngrOff : BOOL ;
   CmdFeedOn : BOOL ;
   CmdFree : BOOL ;
   CmdAutomatic : BOOL ;
   CmdStepOff : BOOL ;
   CmdAutoTolOff : BOOL ;
   CmdDosingMonOn : BOOL ;
   CmdRestDischargeOn : BOOL ;
   CmdScrapBatch : BOOL ;
   Cmd10 : BOOL ;
   Cmd11 : BOOL ;
   Cmd12 : BOOL ;
   Cmd13 : BOOL ;
   Cmd14 : BOOL ;
   Cmd15 : BOOL ;
   CmdSingleIngrOn : BOOL ;
   CmdLogIngrOn : BOOL ;
   CmdFeedOff : BOOL ;
   CmdHold : BOOL ;
   CmdHand : BOOL ;
   CmdStepOn : BOOL ;
   CmdAutoTolOn : BOOL ;
   CmdDosingMonOff : BOOL ;
  END_STRUCT ;	
END_TYPE

TYPE "CWA_UDT_BinParaShort"	// UDT 10418
VERSION : 0.0
  STRUCT 	//UDT for Binparameter short
   BinNr : INT ;
   BinType : STRUCT
    spare0 : BOOL ;
    spare1 : BOOL ;
    spare2 : BOOL ;
    spare3 : BOOL ;
    spare4 : BOOL ;
    spare5 : BOOL ;
    VarBinLL : BOOL ;
    ParModeDosWt : BOOL ;
    ParManualAdd : BOOL ;
    Par1Speed : BOOL ;
    Par2Speed : BOOL ;
    ParFrequency : BOOL ;
   END_STRUCT ;
   VarSwitchOverWtFs : INT ;
   VarCutoffWt : INT ;
   ParTolPosWt : INT  := 15;
   ParTolNegWt : INT  := 10;
   ParCutoffWtCorrMax : INT  := 50;
   ParDosingTimeSlow : INT  := 40;
   ParSwitchOverTime_f_s : INT  := 30;
   ParTipPulseLen : INT  := 5;
   ParDosingTimeMax : INT  := 300;
   ParTolPosPc : INT  := 500;	// (%)
   ParTolNegPc : INT  := 500;	// (%)
   ParTolAutoPosWt : INT ;
   ParTolAutoPosPc : INT ;	// (%)
  END_STRUCT ;	
END_TYPE

TYPE "CWA_UDT_BinParaAll"	// UDT 10419
VERSION : 0.0
  STRUCT 	//UDT for Binparameter full
   BinNr : INT ;
   BinType : STRUCT
    spare0 : BOOL ;
    spare1 : BOOL ;
    spare2 : BOOL ;
    spare3 : BOOL ;
    spare4 : BOOL ;
    spare5 : BOOL ;
    VarBinLL : BOOL ;
    ParModeDosWt : BOOL ;
    ParManualAdd : BOOL ;
    Par1Speed : BOOL ;
    Par2Speed : BOOL ;
    ParFrequency : BOOL ;
   END_STRUCT ;
   VarSwitchOverWtFs : INT ;
   VarCutoffWt : INT ;
   ParTolPosWt : INT  := 15;
   ParTolNegWt : INT  := 10;
   ParCutoffWtCorrMax : INT  := 50;
   ParDosingTimeSlow : INT  := 40;
   ParSwitchOverTime_f_s : INT  := 30;
   ParTipPulseLen : INT  := 5;
   ParDosingTimeMax : INT  := 300;
   ParTolPosPc : INT  := 500;	// (%)
   ParTolNegPc : INT  := 500;	// (%)
   ParTolAutoPosWt : INT ;
   ParTolAutoPosPc : INT ;	// (%)
   ParDosingSpeedFast : INT  := 100;
   ParDosingSpeedSlow : INT  := 20;
   ParFineDosWt : INT  := 50;
   Par19 : INT ;
   Par20 : INT ;
   Par21 : INT ;
  END_STRUCT ;	
END_TYPE

TYPE "GCS7_UDT_FunctionKey"	// UDT 10601
VERSION : 0.0
  STRUCT
   CmdProdCheck : BOOL ;	//ASW: Start after product check
   CmdEmptying : BOOL ;
   CmdTolerate : BOOL ;
   CmdHornOff : BOOL ;
   Cmd04 : BOOL ;
   Cmd05 : BOOL ;
   Cmd06 : BOOL ;
   Cmd07 : BOOL ;
   CmdStart : BOOL ;
   CmdTransferOn : BOOL ;
   CmdFeedOn : BOOL ;
   CmdFree : BOOL ;
   CmdAutomatic : BOOL ;
   CmdStepOff : BOOL ;
   CmdNextStep : BOOL ;
   CmdAcceptSize : BOOL ;
   Cmd16 : BOOL ;
   CmdAbortBatch : BOOL ;
   CmdFaultReset : BOOL ;
   CmdHornOn : BOOL ;
   Cmd17 : BOOL ;
   Cmd18 : BOOL ;
   Cmd19 : BOOL ;
   CmdHLOverride : BOOL ;	//ASW: Activate function override HL
   CmdImmediateStop : BOOL ;
   CmdTransferOff : BOOL ;
   CmdFeedOff : BOOL ;
   CmdHold : BOOL ;
   CmdHand : BOOL ;
   CmdStepOn : BOOL ;
   CmdReset : BOOL ;
   CmdSequenzStop : BOOL ;
  END_STRUCT ;	
END_TYPE

TYPE "GCS7_UDT_FaultPattern"	// UDT 10602
VERSION : 0.0
  STRUCT
   Es00 : BOOL ;
   Es01 : BOOL ;
   Es02 : BOOL ;
   Es03 : BOOL ;
   Es04 : BOOL ;
   Es05 : BOOL ;
   Es06 : BOOL ;
   Es07 : BOOL ;
   Es08 : BOOL ;
   Es09 : BOOL ;
   Es10 : BOOL ;
   Es11 : BOOL ;
   Es12 : BOOL ;
   Es13 : BOOL ;
   Es14 : BOOL ;
   EsNewBinTimeout : BOOL ;	//ASW: Max. delay time to send a new bin
   EsBatchSize : BOOL ;
   EsRefillLevel : BOOL ;
   EsSectionTimeOut : BOOL ;	//ASW: Max. section time to stay in section
   EsHandAddTimeOut : BOOL ;	//ASW: Max. delay time to accept manual ingredients
   EsRecipePlace : BOOL ;	//ASW: Fault recipe place
   EsProductMismatch : BOOL ;	//ASW: Product check failed
   Es22 : BOOL ;
   Es23 : BOOL ;
   EsEmpty : BOOL ;
   EsFull : BOOL ;
   EsWayConflict : BOOL ;
   EsWarning : BOOL ;
   EsMech : BOOL ;
   EsDosing : BOOL ;
   EsEmptying : BOOL ;
   EsInterrupt : BOOL ;
  END_STRUCT ;	
END_TYPE

TYPE "GCS7_UDT_StatusPattern"	// UDT 10603
VERSION : 0.0
  STRUCT
   StaStartRelease : BOOL ;
   StaMixingTime : BOOL ;
   StaMixingTimeEnd : BOOL ;
   Sta03 : BOOL ;
   Sta04 : BOOL ;
   Sta05 : BOOL ;
   Sta06 : BOOL ;
   StaDPFault : BOOL ;
   StaHWStop : BOOL ;
   StaAutostartSec : BOOL ;
   StaAutostart : BOOL ;
   StaOnline : BOOL ;
   StaLoaded : BOOL ;
   StaHandAdd : BOOL ;
   StaEmptyingTime : BOOL ;
   StaStartwarning : BOOL ;
   StaImmediateStopASW : BOOL ;	//ASW: Summary information: Any condition is true
   StaTransferOffASW : BOOL ;	//ASW: Summary information: Any condition is true
   StaFeedOffASW : BOOL ;	//ASW: Summary information: Any condition is true
   Sta23 : BOOL ;
   Sta24 : BOOL ;
   Sta25 : BOOL ;
   Sta26 : BOOL ;
   StaHLOverride : BOOL ;	//ASW: Override function is active
   StaImmediateStop : BOOL ;
   StaTransferOff : BOOL ;
   StaFeedOff : BOOL ;
   StaHold : BOOL ;
   StaHand : BOOL ;
   StaStep : BOOL ;
   StaReset : BOOL ;
   StaEndOfJob : BOOL ;
  END_STRUCT ;	
END_TYPE

TYPE "GCS7_UDT_BINList2"	// UDT 10664
VERSION : 0.0
  STRUCT
   BinNr : INT ;
   InfLocked : BOOL ;
   InfLevelFault : BOOL ;	//Sender empty, Receiver full
   InFeedOff : BOOL ;	//HWStop or DPFault of the connected level probe (*new*)
   OutDryFillingDone : BOOL ;	//Is copied from central bin list
   VarFlagOverwriteLevel : BOOL ;
   InfLowLevel : BOOL ;
   InfLevelMiddle : BOOL ;
   InfHighLevel : BOOL ;
   InfActiveBin : BOOL ;
   InfPreselect : BOOL ;
   InfDeselect : BOOL ;
   spare13 : BOOL ;
   InOutDPFault : BOOL ;	//DP Fault of connected Level
   InfIsInRecipe : BOOL ;	//Bin is used recipe as ingredient
   VarFlagLocked : BOOL ;
   VarFlagLevelFault : BOOL ;
   ParEmptyingTime : INT ;
   WeightActual : DINT ;
   tmpIndex : INT ;	//Index bin in central bin list
  END_STRUCT ;	
END_TYPE

TYPE "GCS7_UDT_BINList3"	// UDT 10668
VERSION : 0.0
  STRUCT
   BinNr : INT ;
   InfLocked : BOOL ;
   InfLevelFault : BOOL ;	//Sender empty, Receiver full
   InFeedOff : BOOL ;	//HWStop or DPFault of the connected level probe (*new*)
   OutDryFillingDone : BOOL ;	//Is copied from central bin list
   VarFlagOverwriteLevel : BOOL ;
   InfLowLevel : BOOL ;
   InfLevelMiddle : BOOL ;
   InfHighLevel : BOOL ;
   InfActiveBin : BOOL ;
   InfPreselect : BOOL ;
   InfDeselect : BOOL ;
   spare13 : BOOL ;
   InOutDPFault : BOOL ;	//DP Fault of connected Level
   InfIsInRecipe : BOOL ;	//Bin is used in recipe as ingredient
   VarFlagLocked : BOOL ;
   VarFlagLevelFault : BOOL ;
   ParEmptyingTime : INT ;
   WeightActual : DINT ;
   WeightTarget : DINT ;
   WeightActualPrev : DINT ;	//Actual weight previous job
   tmpIndex : INT ;	//Index bin in central bin list
  END_STRUCT ;	
END_TYPE

TYPE "GCS7_UDT_ScaleControl"	// UDT 10680
VERSION : 0.0
  STRUCT
   ParScaleInSection : ARRAY  [1 .. 64 ] OF BOOL ;
   ToASW : STRUCT
    spare0 : BOOL ;
    EsRefillLevel : BOOL ;
    CmdTestRefillDone : BOOL ;
    spare3 : BOOL ;
    spare4 : BOOL ;
    spare5 : BOOL ;
    spare6 : BOOL ;
    spare7 : BOOL ;
    InfActive : BOOL ;
    InfEmptying : BOOL ;
    CmdReady : BOOL ;
    CmdEmptied : BOOL ;
    InfFault : BOOL ;
   END_STRUCT ;
   ToSSW : STRUCT
    InfEnableDosing : BOOL ;
    spare1 : BOOL ;
    spare2 : BOOL ;
    spare3 : BOOL ;
    spare4 : BOOL ;
    spare5 : BOOL ;
    spare6 : BOOL ;
    spare7 : BOOL ;
    CmdReset : BOOL ;
    CmdAbortBatch : BOOL ;
    CmdAcceptWt : BOOL ;
    CmdRetry : BOOL ;
   END_STRUCT ;
   CmdStartScale : ARRAY  [1 .. 64 ] OF //Start request for scale 1 to 32
   BOOL ;
   InfActive : ARRAY  [1 .. 64 ] OF //Active Scales
   BOOL ;
   InfEmptied : ARRAY  [1 .. 64 ] OF //Scales which are emptied (finished)
   BOOL ;
  END_STRUCT ;	
END_TYPE

TYPE "ASW_StageCtrl"	// UDT 18000
VERSION : 0.1
  STRUCT
   ToSSW : STRUCT
    CmdStageComplete : BOOL ;
    CmdStageDone : BOOL ;
   END_STRUCT ;
   ToASW : STRUCT
    OutStageEmpty : BOOL ;
    CmdBatchDone : BOOL ;
   END_STRUCT ;
   StageAct : INT ;
   spare11 : INT ;
   spare12 : INT ;
   ScaleUsed : ARRAY  [1 .. 64 ] OF BOOL ;
   ScaleStarted : ARRAY  [1 .. 64 ] OF BOOL ;
   ScaleDone : ARRAY  [1 .. 64 ] OF BOOL ;
   spare8 : INT ;
   spare9 : INT ;
   spare10 : INT ;
  END_STRUCT ;	
END_TYPE

TYPE "WinCoSYieldScale"	// UDT 19001
VERSION : 0.0
  STRUCT
   PCCScaleNo : DINT ;
   JobIdent : DINT ;
   ActualFlowrate : DINT ;
   ActualJobWeight : DINT ;
   NonEraseableWeight : DINT ;
  END_STRUCT ;	
END_TYPE

TYPE "SamplerData"	// UDT 19002
VERSION : 0.0
  STRUCT
   PCCScaleNo : DINT ;
   JobIdent : DINT ;
   ActualFlowrate : DINT ;
   ActualJobWeight : DINT ;
   NonEraseableWeight : DINT ;
  END_STRUCT ;	
END_TYPE

TYPE "GCS7_FB9_Section"	// UDT 20090
VERSION : 0.0
  STRUCT
   All : STRUCT
    CmdClearIdling : BOOL ;	//Stop al groups of this section which are in idling
    OutAutoStartOkShared : BOOL ;	//All multiple used group has autostart bit set
    InASWFlagAutostart : BOOL ;	//Free for ASW
    OutAutostartOkAll : BOOL ;	//Autostart of all selected groups ok
    Spare04 : BOOL ;
    Spare05 : BOOL ;
    OutPreStarted : BOOL ;	//All relevant prestarted groups are started
    OutPreStarting : BOOL ;	//Any group is pre-starting
    Spare10 : BOOL ;
    CmdContinue : BOOL ;	//(*new*)
    CmdManualOffRel : BOOL ;
    CmdFaultReset : BOOL ;	//Command to fault reset
    CmdManualOff : BOOL ;	//Switch off maunual mode of all object
    OutStartwarning : BOOL ;	//Any selected group is in startwarning mode
    OutManualAny : BOOL ;	//Any object of this PLC is in manual mode
    InOutASWSelectionOK : BOOL ;	//Used by ASW
    OutSelectionValid : BOOL ;	//Any object is occupied for this section
    CmdNewSelection : BOOL ;	//An new object is occupied
    OutGrConflict : BOOL ;	//An object is not available
    OutGrIsLocked : BOOL ;	//An object is locked by ASW
    OutAutoStartOk : BOOL ;	//(*new*) All relevant Groups are in mode AutoStart
    OutManual : BOOL ;	//Any object of this section is in manual mode
    OutDPFault : BOOL ;	//(*new*)
    OutHWStop : BOOL ;	//(*new*)
    OutStoppedRel : BOOL ;
    OutStoppedAll : BOOL ;
    OutLoaded : BOOL ;	//(*new*)
    OutFaultIdling : BOOL ;
    OutFaultRel : BOOL ;
    OutFaultAll : BOOL ;
    OutIdling : BOOL ;
    OutWarning : BOOL ;
   END_STRUCT ;
   Feed : STRUCT
    InEnable : BOOL ;
    Spare01 : BOOL ;
    CmdNext : BOOL ;
    Spare03 : BOOL ;
    Spare04 : BOOL ;
    Spare05 : BOOL ;
    Spare06 : BOOL ;
    Spare07 : BOOL ;
    OutStoppedRel : BOOL ;
    OutStoppedAll : BOOL ;
    OutStartedRel : BOOL ;
    OutFaultIdling : BOOL ;
    OutFaultRel : BOOL ;
    OutFaultAll : BOOL ;
    OutIdling : BOOL ;
    OutSelected : BOOL ;
   END_STRUCT ;
   Mgr : STRUCT
    InEnable : BOOL ;
    Spare01 : BOOL ;
    CmdNext : BOOL ;
    Spare03 : BOOL ;
    Spare04 : BOOL ;
    Spare05 : BOOL ;
    Spare06 : BOOL ;
    Spare07 : BOOL ;
    OutStoppedRel : BOOL ;
    OutStoppedAll : BOOL ;
    OutStartedRel : BOOL ;
    OutFaultIdling : BOOL ;
    OutFaultRel : BOOL ;
    OutFaultAll : BOOL ;
    OutIdling : BOOL ;
    OutSelected : BOOL ;
   END_STRUCT ;
   Wgr : STRUCT
    InEnable : BOOL ;
    Spare01 : BOOL ;
    CmdNext : BOOL ;
    Spare03 : BOOL ;
    Spare04 : BOOL ;
    Spare05 : BOOL ;
    Spare06 : BOOL ;
    Spare07 : BOOL ;
    OutStoppedRel : BOOL ;
    OutStoppedAll : BOOL ;
    OutStartedRel : BOOL ;
    OutFaultIdling : BOOL ;
    OutFaultRel : BOOL ;
    OutFaultAll : BOOL ;
    OutIdling : BOOL ;
    OutSelected : BOOL ;
   END_STRUCT ;
   Ggr : STRUCT
    InEnable : BOOL ;
    Spare01 : BOOL ;
    CmdNext : BOOL ;
    Spare03 : BOOL ;
    Spare04 : BOOL ;
    Spare05 : BOOL ;
    Spare06 : BOOL ;
    Spare07 : BOOL ;
    OutStoppedRel : BOOL ;
    OutStoppedAll : BOOL ;
    OutStartedRel : BOOL ;
    OutFaultIdling : BOOL ;
    OutFaultRel : BOOL ;
    OutFaultAll : BOOL ;
    OutIdling : BOOL ;
    OutSelected : BOOL ;
   END_STRUCT ;
   InPreselect : ARRAY  [1 .. 320 ] OF BOOL ;
   OutSelected : ARRAY  [1 .. 320 ] OF BOOL ;
   OutIdling : ARRAY  [1 .. 320 ] OF BOOL ;
   ParNotRelForStarted : ARRAY  [1 .. 320 ] OF BOOL  := FALSE;
   ParNotRelForFault : ARRAY  [1 .. 320 ] OF BOOL  := FALSE;
   InManual : ARRAY  [1 .. 320 ] OF BOOL  := FALSE;
   InPreStart : ARRAY  [1 .. 320 ] OF //Input from section: These groups are pre-starting
   BOOL  := FALSE;
  END_STRUCT ;	
END_TYPE

TYPE "GCS7_GR_COM"	// UDT 20097
VERSION : 0.0
  STRUCT
   SelectedForPLC1 : BOOL ;
   SelectedForPLC2 : BOOL ;
   SelectedForPLC3 : BOOL ;
   SelectedForPLC4 : BOOL ;
   SelectedForPLC5 : BOOL ;
   SelectedForPLC6 : BOOL ;
   SelectedForPLC7 : BOOL ;
   SelectedForPLC8 : BOOL ;
   SelectedForPLC9 : BOOL ;
   SelectedForPLC10 : BOOL ;
   SelectedForPLC11 : BOOL ;
   SelectedForPLC12 : BOOL ;
   SelectedForPLC13 : BOOL ;
   SelectedForPLC14 : BOOL ;
   SelectedForPLC15 : BOOL ;
   SelectedForPLC16 : BOOL ;
   WasSelectedForPLC1 : BOOL ;
   WasSelectedForPLC2 : BOOL ;
   WasSelectedForPLC3 : BOOL ;
   WasSelectedForPLC4 : BOOL ;
   WasSelectedForPLC5 : BOOL ;
   WasSelectedForPLC6 : BOOL ;
   WasSelectedForPLC7 : BOOL ;
   WasSelectedForPLC8 : BOOL ;
   WasSelectedForPLC9 : BOOL ;
   WasSelectedForPLC10 : BOOL ;
   WasSelectedForPLC11 : BOOL ;
   WasSelectedForPLC12 : BOOL ;
   WasSelectedForPLC13 : BOOL ;
   WasSelectedForPLC14 : BOOL ;
   WasSelectedForPLC15 : BOOL ;
   WasSelectedForPLC16 : BOOL ;
   InEnablePLC1 : BOOL ;
   InEnablePLC2 : BOOL ;
   InEnablePLC3 : BOOL ;
   InEnablePLC4 : BOOL ;
   InEnablePLC5 : BOOL ;
   InEnablePLC6 : BOOL ;
   InEnablePLC7 : BOOL ;
   InEnablePLC8 : BOOL ;
   InEnablePLC9 : BOOL ;
   InEnablePLC10 : BOOL ;
   InEnablePLC11 : BOOL ;
   InEnablePLC12 : BOOL ;
   InEnablePLC13 : BOOL ;
   InEnablePLC14 : BOOL ;
   InEnablePLC15 : BOOL ;
   InEnablePLC16 : BOOL ;
   Free : BOOL ;
   MultipleUsed : BOOL ;
   Deselect : BOOL ;
   InEnableGrOld : BOOL ;
  END_STRUCT ;	
END_TYPE

TYPE "GCS90S7_FB9_Communicat"	// UDT 20098
VERSION : 0.1
  STRUCT
   StStopped : BOOL ;	//to virtual group
   StStarting : BOOL ;	//to virtual group
   StStarted : BOOL ;	//to virtual group
   StStopping : BOOL ;	//to virtual group
   StFault : BOOL ;	//to virtual group
   OutWarning : BOOL ;	//to virtual group
   InManual : BOOL ;	//to virtual group
   spare07 : BOOL ;	//to virtual group
   SelectedForPLC1 : BOOL ;	//to virtual group
   SelectedForPLC2 : BOOL ;	//to virtual group
   SelectedForPLC3 : BOOL ;	//to virtual group
   SelectedForPLC4 : BOOL ;	//to virtual group
   MultipleUsed : BOOL ;	//to virtual group
   SelectedForPLC5 : BOOL ;	//to virtual group
   SelectedForPLC6 : BOOL ;	//to virtual group
   ASW17 : BOOL ;	//to virtual group
   InEnableGr : BOOL ;	//to real group
   spare11 : BOOL ;	//to real group
   CmdNext : BOOL ;	//to real group
   CmdFaultReset : BOOL ;	//to real group
   InOccupied : BOOL ;	//to real group
   CmdManualOff : BOOL ;	//to real group
   CmdNewJob : BOOL ;	//to real group
   CmdNewValue : BOOL ;	//to real group
   CmdRestartIdling : BOOL ;	//to real group
   SelectedForPLC7 : BOOL ;	//to virtual group
   SelectedForPLC8 : BOOL ;	//to virtual group
   SelectedForPLC9 : BOOL ;	//to virtual group
   SelectedForPlcX : BOOL ;	//to virtual group : Is selected for this PLC
   ASW35 : BOOL ;	//to real group
   InClose : BOOL ;	//to real group
   InOpen : BOOL ;	//to real group
  END_STRUCT ;	
END_TYPE

TYPE "GCS7_FB9_Communication"	// UDT 20099
VERSION : 0.1
  STRUCT
   StStopped : BOOL ;	//to virtual group
   StStarting : BOOL ;	//to virtual group
   StStarted : BOOL ;	//to virtual group
   StStopping : BOOL ;	//to virtual group
   StFault : BOOL ;	//to virtual group
   OutWarning : BOOL ;	//to virtual group
   InManual : BOOL ;	//to virtual group
   InHWStop : BOOL ;	//to virtual group
   InDPFault : BOOL ;	//to virtual group
   InLoaded : BOOL ;	//to virtual group
   InAutoStart : BOOL ;	//to virtual group
   InStartWarning : BOOL ;	//to virtual group
   SelectedForPLC7 : BOOL ;	//to virtual group
   SelectedForPLC8 : BOOL ;	//to virtual group
   SelectedForPLC1 : BOOL ;	//to virtual group
   SelectedForPLC2 : BOOL ;	//to virtual group
   SelectedForPLC3 : BOOL ;	//to virtual group
   SelectedForPLC4 : BOOL ;	//to virtual group
   MultipleUsed : BOOL ;	//to virtual group
   SelectedForPLC5 : BOOL ;	//to virtual group
   SelectedForPLC6 : BOOL ;	//to virtual group
   StCode : INT ;	//to virtual group
   InEnableGr : BOOL ;	//to real group
   SelectedForPLC9 : BOOL ;	//to real group
   CmdNext : BOOL ;	//to real group
   CmdFaultReset : BOOL ;	//to real group
   InOccupied : BOOL ;	//to real group
   CmdManualOff : BOOL ;	//to real group
   CmdNewJob : BOOL ;	//to real group
   CmdNewValue : BOOL ;	//to real group
   CmdRestartIdling : BOOL ;	//to real group
   CmdContinue : BOOL ;	//to real group
   SelectedForPlcX : BOOL ;	//to real group : Is selected for this PLC
   ASW33 : BOOL ;	//to real group
   ASW34 : BOOL ;	//to real group
   ASW35 : BOOL ;	//to real group
   InClose : BOOL ;	//to real group
   InOpen : BOOL ;	//to real group
  END_STRUCT ;	
END_TYPE

TYPE "GCS7_FB11_Communication"	// UDT 20119
VERSION : 0.1
  STRUCT
   InEnable : BOOL ;	//Enable to run the element (manual and automatic mode)
   spare0201 : BOOL ;
   InContinuous : BOOL ;	//Switch from pulsing signal to continuous signal
   spare0203 : BOOL ;
   spare0204 : BOOL ;
   spare0205 : BOOL ;
   InpRun : BOOL ;	//Only for filter
   InpFaultDev : BOOL ;	//Digital iniput: fault device
   CmdOff : BOOL ;	//Pulse to stop the element immediately (manual mode)
   CmdOn : BOOL ;	//Pulse to start the element (manual mode)
   CmdNext : BOOL ;	//Pulse to start the element in automatic mode (see global flags)
   CmdFaultReset : BOOL ;	//Command to reset fault
   InLocal : BOOL ;	//1= Local mode (no fault by start with service switch)
   InManual : BOOL ;	//1= Manual / 0= Automatic: Set and reset by PC
   InReport : BOOL ;	//Report of all state transitions
   InSeqStop : BOOL ;	//Stop automatically after idling time
   InHWStop : BOOL ;	//HW stop is detected, no fault
   InDPFault : BOOL ;	//DP-Fault is detected, no fault
   OutIdling : BOOL ;	//Idling is active
   OutWarning : BOOL ;	//Delay Time fault is running
   spare0404 : BOOL ;
   spare0405 : BOOL ;
   OutpFaultReset : BOOL ;	//Reset Alarm
   OutpRun : BOOL ;	//Digital output to run element
   StStopped : BOOL ;	//Element is stopped
   StStarting : BOOL ;	//Element is starting
   StStarted : BOOL ;	//Element is started
   spare0503 : BOOL ;
   StFault : BOOL ;	//Element has a fault
   StFalse : BOOL ;	//Element is in local mode and has a fault
   spare0506 : BOOL ;
   OutPausing : BOOL ;	//Pausing time is on (pulsing signal)
  END_STRUCT ;	
END_TYPE

TYPE "GCS7_FB12_Communication"	// UDT 20129
VERSION : 0.1
  STRUCT
   InEnableRev : BOOL ;	//Enable to run the element reverse
   InEnableFwd : BOOL ;	//Enable to run the element forward
   InSlow : BOOL ;	//Speed mode: 1= slow / 0= fast
   InpRunSlow : BOOL ;	//Digital input: 1= element is running slow
   InpRunFast : BOOL ;	//Digital input: 1= element is running fast
   InpRunRev : BOOL ;	//Digital input: 1= element is running reverse
   InpRunFwd : BOOL ;	//Digital input: 1= element is running forward
   InpFaultDev : BOOL ;	//Digital input: 1= overload or fault frequency converter
   CmdOff : BOOL ;	//Pulse to stop the element immediately (manual mode)
   CmdOn : BOOL ;	//Pulse to start the element immediately (manual mode)
   CmdNext : BOOL ;	//Pulse to start the element in automatic mode (see global flags)
   CmdFaultReset : BOOL ;	//Command to reset fault
   InLocal : BOOL ;	//1= Local mode (no fault by start with service switch)
   InManual : BOOL ;	//1= Manual/ 0=Automatic
   InReport : BOOL ;	//Report of all state transitions
   InSeqStop : BOOL ;	//Stop automatically after idling time
   InHWStop : BOOL ;	//HW stop is detected, no fault
   InDPFault : BOOL ;	//DP-Fault is detected, no fault
   OutIdling : BOOL ;	//Idling is active
   OutpRunSlow : BOOL ;	//Digital output to run slow
   OutpRunFast : BOOL ;	//Digital output to run fast
   OutpRunRev : BOOL ;	//Digital output to run reverse
   OutpRunFwd : BOOL ;	//Digital output to run forward
   spare0407 : BOOL ;
   StStopped : BOOL ;	//Element is stopped
   StStarting : BOOL ;	//Element is starting
   StStartedFwd : BOOL ;	//Element is started forward: Next element can start
   StStopping : BOOL ;	//Element is stopping
   StFault : BOOL ;	//Element has a fault
   StStartedRev : BOOL ;	//Element is started reverse: Next Element can start
   InOutManSlow : BOOL ;	//Manual speed mode: 1= slow / 0= fast
   InOutManRev : BOOL ;	//Manual direction mode: 1= reverse / 0= forward
  END_STRUCT ;	
END_TYPE

TYPE "GCS7_FB13_Communication"	// UDT 20139
VERSION : 0.1
  STRUCT
   InEnableLN : BOOL ;	//Target position is LN
   InEnableHN : BOOL ;	//Target position is HN
   spare0202 : BOOL ;
   spare0203 : BOOL ;
   spare0204 : BOOL ;
   InpLN : BOOL ;	//Digital input: limit switch low  position (closed)
   InpHN : BOOL ;	//Digital input: limit switch high position (open)
   InpFaultDev : BOOL ;	//Digital input: fault device
   CmdLN : BOOL ;	//Pulse to set position LN (manual mode)
   CmdHN : BOOL ;	//Pulse to set position HN (manual mode)
   CmdNext : BOOL ;	//Open next element
   CmdFaultReset : BOOL ;	//Command to reset fault
   InLocal : BOOL ;	//1= Local mode (no fault by start with service switch)
   InManual : BOOL ;	//1= Manual/ 0= Automatic
   InReport : BOOL ;	//Report of all state transition
   InSeqStop : BOOL ;	//Stop automatically after idling time
   InHWStop : BOOL ;	//HW stop is detected, no fault
   InDPFault : BOOL ;	//DP-Fault is detected, no fault
   OutIdling : BOOL ;	//Idling time is running
   OutDelayFault : BOOL ;	//Delay time is running
   OutMonFault : BOOL ;	//Monitoring time is running
   OutpLN : BOOL ;	//Digital output: valve low  position (closed)
   OutpHN : BOOL ;	//Digital output: valve high position (open)
   spare0407 : BOOL ;
   StLN : BOOL ;	//Element is in position LN
   StCtoHN : BOOL ;	//Changing to position HN
   StHN : BOOL ;	//Element is in position HN
   StCtoLN : BOOL ;	//Changing to position LN
   StFault : BOOL ;	//Element has a fault (time-out by positioning)
   StNoPosition : BOOL ;	//Element is not in a final position (only in local mode)
  END_STRUCT ;	
END_TYPE

TYPE "GCS7_FB14_Communication"	// UDT 20149
VERSION : 0.1
  STRUCT
   InMonTrue : BOOL ;	//After t4 must be StTrue, otherwise it is a process fault
   InMonFalse : BOOL ;	//After t5 must be StFalse, otherwise it is a process fault
   InPreAlarmTrue : BOOL ;	//LOG Pre-alarm if state is not StTrue
   InPreAlarmFalse : BOOL ;	//LOG Pre-alarm if state is not StFalse
   InStopTrueTime : BOOL ;	//Stop delay time t2
   InStopFalseTime : BOOL ;	//Stop delay time t3
   InpTrue : BOOL ;	//Digital input: signal 'True'; target state is StTrue
   InpFaultDev : BOOL ;	//Digital input: fault device
   CmdRstTrueTime : BOOL ;	//Restart delay time changing from StFalse to StTrue (t2)
   CmdRstFalseTime : BOOL ;	//Restart delay time changing from StTrue to StFalse (t3)
   CmdRunTimeoutTime : BOOL ;	//Run timeout time (only 1 working condition)
   CmdFaultReset : BOOL ;	//Command to reset fault
   InLocal : BOOL ;	//1= Local mode (automatic fault reset)
   spare0305 : BOOL ;	//Copy of InMonTrue to detect change form InMonTrue to InMonFalse
   InReport : BOOL ;	//Report of all state transitions
   OutTimeoutTime : BOOL ;	//Timeout time 1 working condition active
   InHWStop : BOOL ;	//HW stop is detected, no fault
   InDPFault : BOOL ;	//DP-Fault is detected, no fault
   OutPreAlarmTrue : BOOL ;	//Flag PreAlarmTrue is done
   OutPreAlarmFalse : BOOL ;	//Flag PreAlarmFalse is done
   OutFlagPos : BOOL ;	//Positive flag InpTrue
   OutFlagNeg : BOOL ;	//Negative flag InpTrue
   OutpFaultReset : BOOL ;	//Reset alarm
   OutTrue : BOOL ;	//Copy of input signal
   StFalse : BOOL ;	//Signal is 'False', delay time finished, monitoring is off
   StCtoTrue : BOOL ;	//Changing to 'True', signal is 'True'
   StTrue : BOOL ;	//Signal is 'True', delay time finished
   StCtoFalse : BOOL ;	//Changing to 'False', signal is 'False'
   StFault : BOOL ;	//Signal has not requested value, monitoring is active
  END_STRUCT ;	
END_TYPE

TYPE "GCS7_FB16_Communication"	// UDT 20169
VERSION : 0.1
  STRUCT
   InMonMinP : BOOL ;	//Monitoring the minimum pressure
   spare0201 : BOOL ;
   spare0202 : BOOL ;
   spare0203 : BOOL ;
   spare0204 : BOOL ;
   spare0205 : BOOL ;
   InpMin : BOOL ;	//Digital input: Value <= min
   InpMax : BOOL ;	//Digital input: Value >= max
   spare0300 : BOOL ;
   spare0301 : BOOL ;
   spare0302 : BOOL ;
   CmdFaultReset : BOOL ;	//Command to reset fault
   InLocal : BOOL ;	//1= Local mode (no fault by Over Pressure)
   spare0305 : BOOL ;
   InReport : BOOL ;	//Report of all state transition
   spare0307 : BOOL ;
   InHWStop : BOOL ;	//HW stop is detected, no fault
   InDPFault : BOOL ;	//DP-Fault is detected, no fault
   OutNoMinP : BOOL ;	//Warning no minimum pressure
   spare0403 : BOOL ;
   spare0404 : BOOL ;
   spare0405 : BOOL ;
   spare0406 : BOOL ;
   spare0407 : BOOL ;
   StMinP : BOOL ;	//Value <= Minimum
   StNormalP : BOOL ;	//Value in Range Minimum to Maximum
   StOverP : BOOL ;	//Value >= Maximum (only in local mode)
   StCtoOverP : BOOL ;	//Value >= Maximum, delay time is active
   StFault : BOOL ;	//Element has a fault
  END_STRUCT ;	
END_TYPE

TYPE "GCS7_FB37_DP_Alarm"	// UDT 20373
VERSION : 0.1
  STRUCT
   AxxxSoftware : BOOL ;	//A001EPROM, A002RAM, A003RTIM, A004SWDog, A006LostMemory, A079Software
   AxxxCommunication : BOOL ;	//A012HOSTCOM, A014PROFIBUS
   AxxxDisplay : BOOL ;	//A013EXPDISP, W017DISPLAY
   AxxxUnknown : BOOL ;	//Any unknown alarm received
   A005No24V : BOOL ;	//A005 No 24V
   Ax07Range : BOOL ;	//A007 / A107 Signal level is out of range
   A018Battery : BOOL ;	//A018 Batterie
   A024Empty : BOOL ;	//A024 No product for more than 2 minutes
   Ax30Zero : BOOL ;	//A030 / A130 Zero point level is negative
   Ax32ROD : BOOL ;	//A032 / A132 Signal level is not changing
   Ax50FRoll1 : BOOL ;	//A050 / A150 Fault speedmonitor feed roll 1
   Ax51FRoll2 : BOOL ;	//A051 / A151 Fault speedmonitor feed roll 2
   A052RollUp : BOOL ;	//A052 Fault speedmonitor upper rolls
   A053RollLow : BOOL ;	//A053 Fault speedmonitor lower rolls
   A054MotUp : BOOL ;	//A054 Fault motor current upper motor
   A055MotLow : BOOL ;	//A055 Fault motor current lower motor
   A056STBYUP : BOOL ;	//A056 Idle current upper motor to high
   A057STBYDN : BOOL ;	//A057 Idle current lower motor to high
   A058M_Stop : BOOL ;	//A056 Stop button pressed
   A059M_Stop : BOOL ;	//A057 Stop button not released
   Ax60HLInlet : BOOL ;	//A060 / A160 Alarm HL Inlet
   A061HLOut1 : BOOL ;	//A061 Alarm HL Outlet 1
   A062HLOut2 : BOOL ;	//A063 Alarm HL Outlet 2
   A063HLOut3 : BOOL ;	//A063 Alarm HL Outlet 3
   A064HLBackupLeft : BOOL ;	//A064 Alarm HL Backup Left
   W065HLBackupLeft : BOOL ;	//W065 Warning HL Backup Left
   A066HLBackupRight : BOOL ;	//A066 Alarm HL Backup Right
   W067HLBackupRight : BOOL ;	//W067 Warning HL Backup Left
   Ax68InletFull : BOOL ;	//A068 /A168 Alarm Inlet Full
   Ax69DosMax : BOOL ;	//A069 /A169 Maximum speed feed roll
   A070CANCOM : BOOL ;	//A070 Communication fault with can module
   A071CANMOD : BOOL ;	//A071 Fault of any CAN module
   A072CANDOUT : BOOL ;	//A071 Fault of any CAN output signal
   W075WarnTemp : BOOL ;	//W075 Warning temperature > 65 grad
   A076HighTemp : BOOL ;	//A076 Fault temperature > 75 grad
   A077DigOut : BOOL ;	//A077 Alarm Digital outpus
   A078Service : BOOL ;	//A078 Service Mode
   A110Gap : BOOL ;	//A110 Alarm automatically gap control
  END_STRUCT ;	
END_TYPE

TYPE "GCS7_M_FB41_Data"	// UDT 20410
VERSION : 0.0
  STRUCT 	// Interface to maschine FB50
   StCode : INT ;	//State as code
   InEnable : BOOL ;	//Enable to run machine, 0=Immediate stop
   InFeeding : BOOL ;	//Section is feeding
   InLocalWaterControl : BOOL ;	//MOZD uses internal set value
   InRemoteWaterControl : BOOL ;	//MOZD uses set value from PLC
   InManualWaterControl : BOOL ;	//MOZD is bypassed
   CmdNewJob : BOOL ;	//New job
   spare0206 : BOOL ;
   spare0207 : BOOL ;
   CmdOff : BOOL ;	//Pulse to stop all elements immediately (manual mode)
   CmdOn : BOOL ;	//Pusle to start in manual mode
   CmdNext : BOOL ;	//Pulse to start the element in automatic mode (see global flags)
   CmdFaultReset : BOOL ;	//Command to reset fault
   InLocal : BOOL ;	//1= Local mode (no fault by start with service switch)
   InManual : BOOL ;	//1= Manual/ 0=Automatic
   spare0306 : BOOL ;
   spare0307 : BOOL ;
   OutOffDelayFeedRun : BOOL ;	//Aux. signal switch off delay feed is running
   OutOffDelayFeedDone : BOOL ;	//Aux. signal switch off delay feed done
   OutOnDelayWaterRun : BOOL ;	//Aux. signal switch off delay feed done
   OutOnDelayWaterDone : BOOL ;	//Aux. signal switch on delay water done
   spare0404 : BOOL ;
   spare0405 : BOOL ;
   spare0406 : BOOL ;
   OutReadyFeeding : BOOL ;
   StStopped : BOOL ;
   StStarting : BOOL ;
   StStarted : BOOL ;
   StStopping : BOOL ;
   StFault : BOOL ;
   StWaiting : BOOL ;
   Par : STRUCT
    ParObjectNo : INT ;	//Is used for communication with PC
    ParSpare : BOOL  := TRUE;
    ParWithHLInlet : BOOL  := TRUE;	//Machine with element HLInlet
    ParWithAirValve : BOOL  := TRUE;	//Machine with element AirValve
    ParWithBypassFlap : BOOL  := TRUE;	//Machine with element BypassFlap
    ParFlowProdLocal : BOOL ;	//Not ManualWaterControl mode: FlowProd set to local
    ParOffDelayFeed : INT ;	//Switch off delay after feed [0.1 s]
    ParOnDelayWater : INT ;	//Switch on delay for water   [0.1 s]
    OutOffDelayFeed : INT ;	//Actual time: off delay feed timer
    OutOnDelayWater : INT ;	//Actual time: on delay water timer
    spare2000 : INT ;
    spare2200 : INT ;
   END_STRUCT ;
  END_STRUCT ;	
END_TYPE

TYPE "GCS7_M_FB44_Data"	// UDT 20440
VERSION : 0.0
  STRUCT 	// Interface to maschine FB50
   StCode : INT ;	//State as code
   InEnable : BOOL ;	//Enable to run machine
   spare0201 : BOOL ;
   spare0202 : BOOL ;
   spare0203 : BOOL ;
   spare0204 : BOOL ;
   spare0205 : BOOL ;
   spare0206 : BOOL ;
   spare0207 : BOOL ;
   CmdOff : BOOL ;	//Pulse to start the element immediately (manual mode)
   CmdOn : BOOL ;	//Pulse to stop  the element immediately (manual mode)
   CmdNext : BOOL ;	//Pulse to start the element in automatic mode
   CmdFaultReset : BOOL ;	//Command to reset fault
   InLocal : BOOL ;	//1= Local mode (no fault by start with service switch)
   InManual : BOOL ;	//1= Manual/ 0=Automatic
   spare0306 : BOOL ;
   InSeqStop : BOOL ;	//Sequence stop
   spare0400 : BOOL ;
   spare0401 : BOOL ;
   spare0402 : BOOL ;
   spare0403 : BOOL ;
   spare0404 : BOOL ;
   spare0405 : BOOL ;
   spare0406 : BOOL ;
   spare0407 : BOOL ;
   StStopped : BOOL ;
   StStarting : BOOL ;
   StStarted : BOOL ;
   StStopping : BOOL ;
   StFault : BOOL ;
   spare0505 : BOOL ;
   StBypassed : BOOL ;
   Par : STRUCT
    ParObjectNo : INT ;	//Is used for communication with PC
    ParWithAspHigh : BOOL  := TRUE;
    ParWithHL : BOOL  := TRUE;
    ParWithScrew : BOOL ;
    ParWithScraper : BOOL ;
   END_STRUCT ;
  END_STRUCT ;	
END_TYPE

TYPE "GCS7_M_FB45_Data"	// UDT 20450
VERSION : 0.0
  STRUCT 	// Interface to maschine FB50
   StCode : INT ;	//State as code
   InEnable : BOOL ;	//Enable to run machine
   InDisableLeft : BOOL ;	//Left side not used
   InDisableRight : BOOL ;	//Right side not used
   InOverrideHL : BOOL ;
   spare0204 : BOOL ;
   spare0205 : BOOL ;
   InpPressureLeft : BOOL ;	//1=Working pressure rolls
   InpPressureRight : BOOL ;	//1=Working pressure rolls
   CmdOff : BOOL ;	//Pulse to start the element immediately (manual mode)
   CmdOn : BOOL ;	//Pulse to stop  the element immediately (manual mode)
   CmdNext : BOOL ;	//Pulse to start the element in automatic mode
   CmdFaultReset : BOOL ;	//Command to reset fault
   InLocal : BOOL ;	//1= Local mode (no fault by start with service switch)
   InManual : BOOL ;	//1= Manual/ 0=Automatic
   spare0306 : BOOL ;
   InSeqStop : BOOL ;	//Sequence stop
   OutStartupDone : BOOL ;
   OutStartMan : BOOL ;	//Internal used
   spare0402 : BOOL ;
   spare0403 : BOOL ;
   spare0404 : BOOL ;
   spare0405 : BOOL ;
   spare0406 : BOOL ;
   spare0407 : BOOL ;
   StStopped : BOOL ;
   StStarting : BOOL ;
   StStarted : BOOL ;
   StStopping : BOOL ;
   StFault : BOOL ;
   StWarning : BOOL ;
   Par : STRUCT
    ParObjectNo : INT ;	//Is used for communication with PC
    ParWithHLInletLeft : BOOL  := TRUE;
    ParWithHLInletRight : BOOL  := TRUE;
    ParWithSMLeft : BOOL  := TRUE;	//With speedmonitor and Pressure left side
    ParWithSMRight : BOOL  := TRUE;	//With speedmonitor and Pressure right side
    ParWarning : BOOL ;
    ParManual : BOOL ;
   END_STRUCT ;
  END_STRUCT ;	
END_TYPE

TYPE "GCS7_M_FB46_Data"	// UDT 20460
VERSION : 0.0
  STRUCT 	// Interface to maschine FB50
   StCode : INT ;	//State as code
   InEnable : BOOL ;	//Enable to run machine
   InDisableLeft : BOOL ;	//Left side not used
   InDisableRight : BOOL ;	//Right side not used
   InOverwriteHL : BOOL ;
   spare0204 : BOOL ;
   spare0205 : BOOL ;
   InpPressureLeft : BOOL ;	//1=Working pressure rolls
   InpPressureRight : BOOL ;	//1=Working pressure rolls
   CmdOff : BOOL ;	//Pulse to start the element immediately (manual mode)
   CmdOn : BOOL ;	//Pulse to stop  the element immediately (manual mode)
   CmdNext : BOOL ;	//Pulse to start the element in automatic mode
   CmdFaultReset : BOOL ;	//Command to reset fault
   InLocal : BOOL ;	//1= Local mode (no fault by start with service switch)
   InManual : BOOL ;	//1= Manual/ 0=Automatic
   spare0306 : BOOL ;
   InSeqStop : BOOL ;	//Sequence stop
   OutStartupDone : BOOL ;
   OutStartMan : BOOL ;	//Internal used
   spare0402 : BOOL ;
   spare0403 : BOOL ;
   spare0404 : BOOL ;
   spare0405 : BOOL ;
   spare0406 : BOOL ;
   spare0407 : BOOL ;
   StStopped : BOOL ;
   StStarting : BOOL ;
   StStarted : BOOL ;
   StStopping : BOOL ;
   StFault : BOOL ;
   StWarning : BOOL ;
   Par : STRUCT
    ParObjectNo : INT ;	//Is used for communication with PC
    ParWithHLInletLeft : BOOL  := TRUE;
    ParWithHLInletRight : BOOL  := TRUE;
    ParWithSMLeft : BOOL  := TRUE;	//With speedmonitor and Pressure left side
    ParWithSMRight : BOOL  := TRUE;	//With speedmonitor and Pressure right side
    ParWarning : BOOL ;
    ParManual : BOOL ;
    Par4Rolls : BOOL ;
   END_STRUCT ;
  END_STRUCT ;	
END_TYPE

TYPE "GCS7_M_FB47_Data"	// UDT 20470
VERSION : 0.0
  STRUCT 	// Interface to maschine FB50
   StCode : INT ;	//State as code
   InEnable : BOOL ;	//Enable to run machine
   InMiddle1 : BOOL ;	//Target position for slide is StMiddle1
   InMiddle2 : BOOL ;	//Target position for slide is StMiddle2
   InFullOpen : BOOL ;	//Target position for slide is StHN
   InEmptying : BOOL ;	//Completly discharge cooler
   CmdRestdischarge : BOOL ;	//Command to finally discharge in state StEmptying
   spare0206 : BOOL ;
   spare0207 : BOOL ;
   CmdOff : BOOL ;	//Pulse to start the element immediately (manual mode)
   CmdOn : BOOL ;	//Pulse to stop  the element immediately (manual mode)
   CmdNext : BOOL ;	//Pulse to start the element in automatic mode
   CmdFaultReset : BOOL ;	//Command to reset fault
   InLocal : BOOL ;	//1= Local mode (no fault by start with service switch)
   InManual : BOOL ;	//1= Manual/ 0=Automatic
   spare0306 : BOOL ;
   spare0307 : BOOL ;
   OutEmptyingTimeDone : BOOL ;	//Wait for command CmdRestDischarge
   OutRestDischarge : BOOL ;	//Slide is moving to StHN
   spare0402 : BOOL ;
   spare0403 : BOOL ;
   spare0404 : BOOL ;
   spare0405 : BOOL ;
   spare0406 : BOOL ;
   spare0407 : BOOL ;
   StStopped : BOOL ;
   StStarting : BOOL ;
   StStarted : BOOL ;
   StStopping : BOOL ;
   StFault : BOOL ;
   StEmptying : BOOL ;
   StEmptied : BOOL ;
   Par : STRUCT
    ParObjectNo : INT ;	//Is used for communication with PC
    ParWithLevel : BOOL  := TRUE;	//With element
    ParAutoRestDischarge : BOOL  := TRUE;	//Do not wait for CmdRestDischarge
    ParEmptyingTime : INT ;	//[0.1s]
    OutEmptyingTime : INT ;	//[0.1s]
    spare8 : INT ;
   END_STRUCT ;
  END_STRUCT ;	
END_TYPE

TYPE "GCS7_M_FB48_Data"	// UDT 20480
VERSION : 0.0
  STRUCT 	// Interface to maschine FB50
   StCode : INT ;	//State as code
   InEnable : BOOL ;	//Enable to run machine
   InDisableM2 : BOOL ;	//Stop motor 2 and 3
   InDisableM3 : BOOL ;	//Stop motor 3
   spare0203 : BOOL ;
   spare0204 : BOOL ;
   spare0205 : BOOL ;
   spare0206 : BOOL ;
   spare0207 : BOOL ;
   CmdOff : BOOL ;	//Pulse to start the element immediately (manual mode)
   CmdOn : BOOL ;	//Pulse to stop  the element immediately (manual mode)
   CmdNext : BOOL ;	//Pulse to start the element in automatic mode
   CmdFaultReset : BOOL ;	//Command to reset fault
   InLocal : BOOL ;	//1= Local mode (no fault by start with service switch)
   InManual : BOOL ;	//1= Manual/ 0=Automatic
   spare0306 : BOOL ;
   InSeqStop : BOOL ;	//Sequence stop
   spare0400 : BYTE ;
   StStopped : BOOL ;
   StStarting : BOOL ;
   StStarted : BOOL ;
   StStopping : BOOL ;
   StFault : BOOL ;
   Par : STRUCT
    ParObjectNo : INT ;	//Is used for communication with PC
    ParWithMotor3 : BOOL  := TRUE;
    ParWithHLLow : BOOL  := TRUE;
    ParWithHLInlet : BOOL  := TRUE;
    ParMotor1IsFan : BOOL ;	//Motor1 stops after idling time
    ParTypeSeparator : BOOL ;	//Start Motor2-->Motor1-->Motor3,No interlocking Motor2 and Motor3
    ParWithScraper : BOOL ;
   END_STRUCT ;
  END_STRUCT ;	
END_TYPE

TYPE "GCS7_M_FB49_Data"	// UDT 20490
VERSION : 0.0
  STRUCT 	// Interface to maschine FB50
   StCode : INT ;	//State as code
   InEnable : BOOL ;	//Enable to run machine
   InEnableEngage : BOOL ;	//Signal to engage the rolls
   InRestdischarge : BOOL ;	//Signal to activate restdischarge mode
   InOverrideHL : BOOL ;	//Override HL (for start up)
   spare0204 : BOOL ;
   spare0205 : BOOL ;
   spare0206 : BOOL ;
   spare0207 : BOOL ;
   CmdOff : BOOL ;	//Pulse to start the element immediately (manual mode)
   CmdOn : BOOL ;	//Pulse to stop  the element immediately (manual mode)
   CmdNext : BOOL ;	//Pulse to start the element in automatic mode
   CmdFaultReset : BOOL ;	//Command to reset fault
   InLocal : BOOL ;	//1= Local mode (no fault by start with service switch)
   InManual : BOOL ;	//1= Manual/ 0=Automatic
   spare0306 : BOOL ;
   InSeqStop : BOOL ;	//Sequence stop
   OutStartupDone : BOOL ;	//Ready to start next roll stand
   OutStartMan : BOOL ;	//Internal used
   spare0402 : BOOL ;
   spare0403 : BOOL ;
   spare0404 : BOOL ;
   spare0405 : BOOL ;
   spare0406 : BOOL ;
   spare0407 : BOOL ;
   StStopped : BOOL ;	//All motors are stopped
   StStarting : BOOL ;	//Not all relevant motors are started
   StStarted : BOOL ;	//All used motors are started
   StStopping : BOOL ;	//Any motor is stopping
   StFault : BOOL ;	//Any relevant element has a fault
   StWarning : BOOL ;	//Any motor has a fault (ParWarning) or any el. is in warning
   Par : STRUCT
    ParObjectNo : INT ;	//Is used for communication with PC
    ParWithRollsLow : BOOL ;	//With motor rolls low
    ParWithHLInlet : BOOL  := TRUE;	//With HL inlet
    ParWithHLBackUp : BOOL ;	//With HL backup
    ParWithHLOutlet : BOOL  := TRUE;	//With HL outlet
    ParWarning : BOOL ;	//Warning mode
    ParManual : BOOL ;	//No interlocking in manual mode
    ParWithCollectAlarm : BOOL ;	//With collected alarm input
    ParWithMddLC : BOOL ;	//With MDDx local control unit (serial communication)
    ParWithFU_FeedRoll : BOOL ;	//With FU Feedroll
    ParB1 : BOOL ;	//B1 roller mill
   END_STRUCT ;
  END_STRUCT ;	
END_TYPE

TYPE "GCS7_M_FB50_Data"	// UDT 20500
VERSION : 0.0
  STRUCT 	// Interface to maschine FB50
   StCode : INT ;	//State as code
   InEnableRev : BOOL ;	//Enable to run the motor reverse
   InEnableFwd : BOOL ;	//Enable to run the motor forward
   InOverrideHLOutlet : BOOL ;	//Ignor HL outlet =Mon1
   spare0203 : BOOL ;
   OutEdgeFaultReset : BOOL ;	//Internal used to detect positve edge of CmdFaultReset
   OutFaultResetFcttst : BOOL ;	//Fault reset after function test
   InpControlEBM : BOOL ;
   InpLocked : BOOL ;	//Machine is not available
   CmdOff : BOOL ;	//Pulse to stop motor immediately in manual mode
   CmdOn : BOOL ;	//Pulse to start in manual mode
   CmdNext : BOOL ;	//Pulse to start the element in automatic mode
   CmdFaultReset : BOOL ;	//Command to reset fault
   InLocal : BOOL ;	//1= Local mode (no fault by start with service switch)
   InManual : BOOL ;	//1= Manual/ 0=Automatic
   CmdTestEBM : BOOL ;	//Pulse to start the test sequence for EBM   [7.0]
   InSeqStop : BOOL ;	//Stop automatically after idling time
   OutWarning : BOOL ;	//Warning Element HlInlet not in StTrue
   InfBMTopOk : BOOL ;	//function ok BM Top                         [7.0]
   InfBMBottomOk : BOOL ;	//function ok BM Bottom                      [7.0]
   InfSMOk : BOOL ;	//function ok SM                             [7.0]
   OutpFcttst_BM_Top : BOOL ;	//Output test BM Top active                  [7.0]
   OutpFcttst_BM_Bottom : BOOL ;	//Output test BM bottom active               [7.0]
   OutpFcttst_SM : BOOL ;	//Output test SM active                      [7.0]
   OutpFaultReset : BOOL ;	//Reset alarm                                [7.0]
   StStopped : BOOL ;	//Motor is stopped
   StStarting : BOOL ;	//Motor is starting
   StStartedFwd : BOOL ;	//Motor is started forward: Next Element can start
   StStopping : BOOL ;	//Motor is stopping
   StFault : BOOL ;	//Machine has a fault
   StStartedRev : BOOL ;	//Machine is started reverse: Next Element can start
   StLocked : BOOL ;	//Machine is external locked
   OutTestTime : INT ;	//time to the next test in s                 [7.0]
   Par : STRUCT
    ParObjectNo : INT ;	//Is used for communication with PC
    ParWithMon1 : BOOL  := TRUE;	//With monitoring element Mon1               [7.0]
    ParWithMon3 : BOOL  := TRUE;	//With monitoring element Mon3
    ParWithMon4 : BOOL  := TRUE;	//With monitoring element Mon4
    ParWithMon5 : BOOL  := TRUE;	//With monitoring element Mon5               [7.0]
    ParWithMon6 : BOOL  := TRUE;	//With monitoring element Mon6               [7.0]
    ParMon1IsHL : BOOL ;	//Mon1 is a high level
    ParMon1IsLS : BOOL ;	//Mon1 is controlled a limit switch
    ParMon1StopByFault : BOOL  := TRUE;	//Mon1 stops motor by fault
    ParMon2IsLS : BOOL ;	//Mon2 is controlled a limit switch
    ParMon3IsLS : BOOL ;	//Mon3 is controlled a limit switch
    ParMon4AsWarning : BOOL ;	//Mon4 is only a Warning Element
    ParMon4StopByFault : BOOL ;	//Mon4 stops motor by fault
    ParMon4IsLS : BOOL ;	//Mon4 is controlled a limit switch
    ParEBM : BOOL  := TRUE;	//With monitoring EBM (elevator fault monitor) [7.0]
    ParMon4IsSM : BOOL ;	//Mon4 is SM
   END_STRUCT ;
  END_STRUCT ;	
END_TYPE

TYPE "GCS7_M_FB51_Data"	// UDT 20510
VERSION : 0.0
  STRUCT 	// Interface to maschine FB50
   StCode : INT ;	//State as code
   InEnableRev : BOOL ;	//Enable to run the motor reverse
   InEnableFwd : BOOL ;	//Enable to run the motor forward
   spare02 : BOOL ;
   spare03 : BOOL ;
   spare04 : BOOL ;
   spare05 : BOOL ;
   spare06 : BOOL ;
   spare07 : BOOL ;
   CmdOff : BOOL ;	//Pulse to stop the machine in manual mode
   CmdOn : BOOL ;	//Pulse to start machine in manual mode
   CmdNext : BOOL ;	//Pulse to start the element in automatic mode
   CmdFaultReset : BOOL ;	//Command to reset fault
   InLocal : BOOL ;	//1= Local mode (no fault by start with service switch)
   InManual : BOOL ;	//1= Manual/ 0=Automatic
   spare16 : BOOL ;
   InSeqStop : BOOL ;	//Stop automatically after idling time
   OutWarning : BOOL ;	//Mon1 is NOT in state StTrue (only with pre-alarm)
   spare0401 : BOOL ;
   spare0402 : BOOL ;
   spare0403 : BOOL ;
   spare0404 : BOOL ;
   spare0405 : BOOL ;
   spare0406 : BOOL ;
   spare0407 : BOOL ;
   StStopped : BOOL ;	//Motor is stopped
   StStarting : BOOL ;	//Motor is starting
   StStartedFwd : BOOL ;	//Motor is started forward: Next Element can start
   StStopping : BOOL ;	//Motor is stopping
   StFault : BOOL ;	//Machine has a fault
   StStartedRev : BOOL ;	//Machine is started reverse: Next Element can start
   Par : STRUCT
    ParObjectNo : INT ;	//Is used for communication with PC
    ParWithMon1 : BOOL  := TRUE;	//With monitoring element Mon1
    ParWithMon2 : BOOL  := TRUE;	//With monitoring element Mon2
    ParMon1IsLS : BOOL ;	//Mon1 is a limit switch
    ParMon1PreAlarm : BOOL ;	//Mon1 activate pre alarm function
    ParMon1StopByFault : BOOL ;	//Mon1 stops motor by fault
    ParMon2IsLS : BOOL ;	//Mon2 is a limit switch
    ParMon2IsHL : BOOL ;	//Mon2 is a high level inlet
    ParMon2NoFault : BOOL ;	//Mon2 makes no fault (no alarm)
    ParMon2StopByFault : BOOL ;	//Mon2 stops motor by fault
    ParMon1IsPS : BOOL ;	//Mon1 is a pressure switch (1 working condition)
   END_STRUCT ;
  END_STRUCT ;	
END_TYPE

TYPE "GCS7_M_FB52_Data"	// UDT 20520
VERSION : 0.0
  STRUCT 	// Interface to maschine FB50
   StCode : INT ;	//State as code
   InEnableRev : BOOL ;	//Enable to run the motor reverse
   InEnableFwd : BOOL ;	//Enable to run the motor forward
   InBypass : BOOL ;	//Machine must set flap VLS1 to position bypassed
   InBypass2 : BOOL ;	//Machine must set flap VLS2 to position bypassed
   InPressureOK : BOOL ;	//Only Machine mit Seal
   spare0205 : BOOL ;
   spare0206 : BOOL ;
   spare0207 : BOOL ;
   CmdOff : BOOL ;	//Pulse to stop the machine in manual mode
   CmdOn : BOOL ;	//Pulse to start machine in manual mode
   CmdNext : BOOL ;	//Pulse to start the element in automatic mode
   CmdFaultReset : BOOL ;	//Command to reset fault
   InLocal : BOOL ;	//1= Local mode (no fault by start with service switch)
   InManual : BOOL ;	//1= Manual/ 0=Automatic
   spare16 : BOOL ;
   InSeqStop : BOOL ;	//Stop automatically after idling time
   OutStartReq : BOOL ;	//Start of motor is requested
   spare0401 : BOOL ;
   spare0402 : BOOL ;
   spare0403 : BOOL ;
   spare0404 : BOOL ;
   spare0405 : BOOL ;
   spare0406 : BOOL ;
   spare0407 : BOOL ;
   StStopped : BOOL ;	//Motor is stopped
   StStarting : BOOL ;	//Motor is starting
   StStarted : BOOL ;	//Motor is startedt
   StStopping : BOOL ;	//Motor is stopping
   StFault : BOOL ;	//Machine has a fault
   StClearing : BOOL ;	//Clearing time is running
   StBypassed : BOOL ;	//Maschine is bypassed,Motor stopped
   Par : STRUCT
    ParObjectNo : INT ;	//Is used for communication with PC
    ParWithMon1 : BOOL  := TRUE;	//With element Mon1
    ParWithHLInlet : BOOL  := TRUE;	//With element HL inlet
    ParMon1IsLS : BOOL ;	//Mon1 is a limit switch
    ParMon1IsHL : BOOL ;	//Mon1 is a high level
    ParMon1StopByFault : BOOL  := TRUE;	//Mon1 stops motor by fault
    ParLocalPosition : BOOL ;	//Manual flap:Use actual position as target position
    ParWithVLS2 : BOOL ;	//With element VLS2
    ParWithSeal : BOOL ;	//With element Seal
    ParClearingTime : INT  := 50;	//Clearing time by deselect motor befor stop
    OutClearingTime : INT ;	//Actual clearing time
    spare8 : INT ;
   END_STRUCT ;
  END_STRUCT ;	
END_TYPE

TYPE "GCS7_M_FB53_Data"	// UDT 20530
VERSION : 0.0
  STRUCT 	// Interface to maschine FB50
   StCode : INT ;	//State as code
   InEnableOpen : BOOL ;	//Enable to run open
   InDisableVibro : BOOL ;	//Disable Vibro
   spare0202 : BOOL ;
   spare0203 : BOOL ;
   spare0204 : BOOL ;
   spare0205 : BOOL ;
   spare0206 : BOOL ;
   spare0207 : BOOL ;
   CmdClose : BOOL ;	//Pulse to close in manual mode
   CmdOpen : BOOL ;	//Pulse to open  in manual mode
   CmdNext : BOOL ;	//Pulse to start the element in automatic mode
   CmdFaultReset : BOOL ;	//Command to reset fault
   InLocal : BOOL ;	//1= Local mode (no fault by start with service switch)
   InManual : BOOL ;	//1= Manual/ 0=Automatic
   spare0306 : BOOL ;
   spare0307 : BOOL ;
   OutDisableRead : BOOL ;	//Any element is moveing, don't read scale value
   OutOpenManReq : BOOL ;	//Manual open requested
   OutPulseClose : BOOL ;	//Pulse closing
   spare0403 : BOOL ;
   spare0404 : BOOL ;
   spare0405 : BOOL ;
   spare0406 : BOOL ;
   spare0407 : BOOL ;
   StClosed : BOOL ;	//Hopper is closed
   StOpening : BOOL ;	//Hopper is opening
   StOpen : BOOL ;	//Hopper is open
   StClosing : BOOL ;	//Hopper is closing
   StFault : BOOL ;	//Any elelemt has a fault
   Par : STRUCT
    ParObjectNo : INT ;	//Is used for communication with PC
    ParWithAirFlap : BOOL  := TRUE;	//With element air recycling flap
    ParWithVLSLower : BOOL  := TRUE;	//With element VLSLower
    ParWithVLSUpper : BOOL  := TRUE;	//With element VLSUpper
    ParWithVibro : BOOL  := TRUE;	//With element Vibro
    ParPulsing : BOOL ;	//Upper flap is pulsing durig emptying
    ParVibroIsMotor : BOOL ;	//Type of Vibro is FB12
    ParWithAirFlap2 : BOOL ;	//With 2 element air recycling flap [5.0]
    ParPulseClosing : INT  := 5;	//By pulsing flap:Pulse length closing [0.1s]
    ParWaitOpen : INT  := 20;	//By pulsing flap:Waiting time in position open [0.1s]
    OutTime : INT ;	//Actual time
   END_STRUCT ;
  END_STRUCT ;	
END_TYPE

TYPE "GCS7_M_FB54_Data"	// UDT 20540
VERSION : 0.0
  STRUCT 	// Interface to maschine FB50
   StCode : INT ;	//State as code
   InEnable : BOOL ;	//Enable to run the motor
   InRunPreMix : BOOL ;	//Enable run premix time
   InRunMainMix : BOOL ;	//Enable run main mix time
   InOpen : BOOL ;	//Mixer is open
   spare04 : BOOL ;
   spare05 : BOOL ;
   spare06 : BOOL ;
   CmdNewBatch : BOOL ;	//New batch in mixer
   CmdOff : BOOL ;	//Pulse to stop the machine in manual mode
   CmdOn : BOOL ;	//Pulse to start machine in manual mode
   CmdNext : BOOL ;	//Pulse to start the element in automatic mode
   CmdFaultReset : BOOL ;	//Command to reset fault
   InLocal : BOOL ;	//1= Local mode (no fault by start with service switch)
   InManual : BOOL ;	//1= Manual/ 0=Automatic
   spare16 : BOOL ;
   InSeqStop : BOOL ;	//Stop automatically after idling time
   OutPreMixIsOn : BOOL ;	//Pre mixing time is on
   OutPreMixDone : BOOL ;	//Pre mixing time finished
   OutMainMixIsOn : BOOL ;	//Main mixing time is on
   OutMainMixDone : BOOL ;	//Main mixing time finished
   OutAfterMixIsOn : BOOL ;	//After mixing time is on
   OutAfterMixDone : BOOL ;	//After mixing time is finished
   OutEmptied : BOOL ;	//Mixer is emptied
   spare0407 : BOOL ;
   StStopped : BOOL ;	//Motor is stopped
   StStarting : BOOL ;	//Motor is starting
   StStarted : BOOL ;	//Motor is started
   StStopping : BOOL ;	//Motor is stopping
   StFault : BOOL ;	//Machine has a fault
   InPreMixTime : INT ;	//Target pre-mix time
   InMainMixTime : INT ;	//Target main-mix time
   OutMixTime : INT ;	//Actual time of actual step
   Par : STRUCT
    ParObjectNo : INT ;	//Is used for communication with PC
    ParWithMon1 : BOOL  := TRUE;	//With element Mon1
    ParWithMon2 : BOOL  := TRUE;	//With element Mon2
    ParMon2IsLS : BOOL ;	//Mon2 is a limit switch
    ParAfterMixTime : INT  := 300;	//Maximum over mix time before stop motor
    spare6 : INT ;
    spare8 : INT ;
   END_STRUCT ;
  END_STRUCT ;	
END_TYPE

